LIN {X 0,Y 573.207,Z 132.087,A -85,B 0,C 180,E1 -2272.999,E2 -2272.999} C_VEL
LIN {X 0,Y 573.202,Z 132.089,A -85,B 0,C 180,E1 -2275.413,E2 -2275.413} C_VEL
LIN {X 0,Y 573.193,Z 132.083,A -85,B 0,C 180,E1 -2278.017,E2 -2278.017} C_VEL
LIN {X 0,Y 573.202,Z 132.084,A -85,B 0,C 180,E1 -2280.877,E2 -2280.877} C_VEL
LIN {X 0,Y 573.19,Z 132.087,A -85,B 0,C 180,E1 -2283.513,E2 -2283.513} C_VEL
LIN {X 0,Y 573.177,Z 132.082,A -85,B 0,C 180,E1 -2286.055,E2 -2286.055} C_VEL
LIN {X 0,Y 573.175,Z 132.086,A -85,B 0,C 180,E1 -2288.707,E2 -2288.707} C_VEL
LIN {X 0,Y 573.185,Z 132.084,A -85,B 0,C 180,E1 -2291.588,E2 -2291.588} C_VEL
LIN {X 0,Y 573.207,Z 132.08,A -85,B 0,C 180,E1 -2294.337,E2 -2294.337} C_VEL
LIN {X 0,Y 573.21,Z 132.082,A -85,B 0,C 180,E1 -2297.362,E2 -2297.362} C_VEL
LIN {X 0,Y 573.22,Z 132.081,A -85,B 0,C 180,E1 -2300.572,E2 -2300.572} C_VEL
LIN {X 0,Y 573.221,Z 132.083,A -85,B 0,C 180,E1 -2303.075,E2 -2303.075} C_VEL
LIN {X 0,Y 573.222,Z 132.077,A -85,B 0,C 180,E1 -2305.668,E2 -2305.668} C_VEL
LIN {X 0,Y 573.209,Z 132.079,A -85,B 0,C 180,E1 -2308.182,E2 -2308.182} C_VEL
LIN {X 0,Y 573.215,Z 132.086,A -85,B 0,C 180,E1 -2310.631,E2 -2310.631} C_VEL
LIN {X 0,Y 573.197,Z 132.08,A -85,B 0,C 180,E1 -2313.517,E2 -2313.517} C_VEL
LIN {X 0,Y 573.191,Z 132.082,A -85,B 0,C 180,E1 -2316.133,E2 -2316.133} C_VEL
LIN {X 0,Y 573.219,Z 132.077,A -85,B 0,C 180,E1 -2319.172,E2 -2319.172} C_VEL
LIN {X 0,Y 573.198,Z 132.084,A -85,B 0,C 180,E1 -2322.15,E2 -2322.15} C_VEL
LIN {X 0,Y 573.213,Z 132.078,A -85,B 0,C 180,E1 -2325.08,E2 -2325.08} C_VEL
LIN {X 0,Y 573.226,Z 132.079,A -85,B 0,C 180,E1 -2327.97,E2 -2327.97} C_VEL
LIN {X 0,Y 573.202,Z 132.084,A -85,B 0,C 180,E1 -2330.116,E2 -2330.116} C_VEL
LIN {X 0,Y 573.225,Z 132.076,A -85,B 0,C 180,E1 -2332.958,E2 -2332.958} C_VEL
LIN {X 0,Y 573.273,Z 132.07,A -85,B 0,C 180,E1 -2335.077,E2 -2335.077} C_VEL
LIN {X 0,Y 573.309,Z 132.07,A -85,B 0,C 180,E1 -2337.892,E2 -2337.892} C_VEL
LIN {X 0,Y 573.32,Z 132.071,A -85,B 0,C 180,E1 -2340,E2 -2340} C_VEL
LIN {X 0,Y 573.274,Z 132.071,A -85,B 0,C 180,E1 -2342.811,E2 -2342.811} C_VEL
LIN {X 0,Y 573.268,Z 132.074,A -85,B 0,C 180,E1 -2345.628,E2 -2345.628} C_VEL
LIN {X 0,Y 573.238,Z 132.077,A -85,B 0,C 180,E1 -2348.46,E2 -2348.46} C_VEL
LIN {X 0,Y 573.241,Z 132.076,A -85,B 0,C 180,E1 -2351.313,E2 -2351.313} C_VEL
LIN {X 0,Y 573.247,Z 132.076,A -85,B 0,C 180,E1 -2354.408,E2 -2354.408} C_VEL
LIN {X 0,Y 573.197,Z 132.081,A -85,B 0,C 180,E1 -2357.114,E2 -2357.114} C_VEL
LIN {X 0,Y 573.205,Z 132.083,A -85,B 0,C 180,E1 -2360.078,E2 -2360.078} C_VEL
LIN {X 0,Y 573.2,Z 132.081,A -85,B 0,C 180,E1 -2362.339,E2 -2362.339} C_VEL
LIN {X 0,Y 573.199,Z 132.081,A -85,B 0,C 180,E1 -2364.344,E2 -2364.344} C_VEL
LIN {X 0,Y 572.561,Z 132.161,A -85,B 0,C 180,E1 -2364.93,E2 -2364.93} C_VEL
LIN {X 0,Y 569.729,Z 132.519,A -85,B 0,C 180,E1 -2365.882,E2 -2365.882} C_VEL
LIN {X 0,Y 567.308,Z 132.823,A -85,B 0,C 180,E1 -2366.648,E2 -2366.648} C_VEL
LIN {X 0,Y 566.25,Z 132.952,A -85,B 0,C 180,E1 -2367.239,E2 -2367.239} C_VEL
LIN {X 0,Y 566.155,Z 132.962,A -85,B 0,C 180,E1 -2367.439,E2 -2367.439} C_VEL
LIN {X 0,Y 566.153,Z 132.964,A -85,B 0,C 180,E1 -2369.772,E2 -2369.772} C_VEL
LIN {X 0,Y 566.195,Z 132.953,A -85,B 0,C 180,E1 -2372.428,E2 -2372.428} C_VEL
LIN {X 0,Y 566.168,Z 132.959,A -85,B 0,C 180,E1 -2374.987,E2 -2374.987} C_VEL
LIN {X 0,Y 566.213,Z 132.958,A -85,B 0,C 180,E1 -2377.909,E2 -2377.909} C_VEL
LIN {X 0,Y 566.226,Z 133.057,A -85,B 0,C 180,E1 -2378.247,E2 -2378.247} C_VEL
LIN {X 0,Y 566.536,Z 138.801,A -85,B 0,C 180,E1 -2379.247,E2 -2379.247} C_VEL
LIN {X 0,Y 566.37,Z 154.943,A -85,B 0,C 180,E1 -2382.073,E2 -2382.073} C_VEL
LIN {X 0,Y 566.258,Z 166.155,A -85,B 0,C 180,E1 -2384.046,E2 -2384.046} C_VEL
LIN {X 0,Y 567.19,Z 172.386,A -85,B 0,C 180,E1 -2384.155,E2 -2384.155} C_VEL
LIN {X 0,Y 566.959,Z 273.025,A -85,B 0,C 180,E1 -2385.45,E2 -2385.45} C_VEL
LIN {X 0,Y 566.865,Z 286.291,A -85,B 0,C 180,E1 -2385.767,E2 -2385.767} C_VEL
LIN {X 0,Y 566.74,Z 298.58,A -85,B 0,C 180,E1 -2386.202,E2 -2386.202} C_VEL
LIN {X 0,Y 566.586,Z 310.977,A -85,B 0,C 180,E1 -2386.799,E2 -2386.799} C_VEL
LIN {X 0,Y 566.444,Z 321.518,A -85,B 0,C 180,E1 -2387.453,E2 -2387.453} C_VEL
LIN {X 0,Y 566.316,Z 331.988,A -85,B 0,C 180,E1 -2388.258,E2 -2388.258} C_VEL
LIN {X 0,Y 566.172,Z 340.62,A -85,B 0,C 180,E1 -2389.069,E2 -2389.069} C_VEL
LIN {X 0,Y 566.099,Z 349.526,A -85,B 0,C 180,E1 -2390.089,E2 -2390.089} C_VEL
LIN {X 0,Y 565.996,Z 356.78,A -85,B 0,C 180,E1 -2391.117,E2 -2391.117} C_VEL
LIN {X 0,Y 565.951,Z 363.434,A -85,B 0,C 180,E1 -2392.295,E2 -2392.295} C_VEL
LIN {X 0,Y 565.918,Z 368.346,A -85,B 0,C 180,E1 -2393.409,E2 -2393.409} C_VEL
LIN {X 0,Y 565.882,Z 372.568,A -85,B 0,C 180,E1 -2394.698,E2 -2394.698} C_VEL
LIN {X 0,Y 565.858,Z 375.371,A -85,B 0,C 180,E1 -2396.02,E2 -2396.02} C_VEL
LIN {X 0,Y 565.827,Z 376.461,A -85,B 0,C 180,E1 -2396.872,E2 -2396.872} C_VEL
LIN {X 0,Y 565.854,Z 376.934,A -85,B 0,C 180,E1 -2397.719,E2 -2397.719} C_VEL
LIN {X 0,Y 565.863,Z 376.636,A -85,B 0,C 180,E1 -2398.979,E2 -2398.979} C_VEL
LIN {X 0,Y 565.878,Z 374.842,A -85,B 0,C 180,E1 -2400.387,E2 -2400.387} C_VEL
LIN {X 0,Y 565.895,Z 372.452,A -85,B 0,C 180,E1 -2401.436,E2 -2401.436} C_VEL
LIN {X 0,Y 565.938,Z 368.487,A -85,B 0,C 180,E1 -2402.646,E2 -2402.646} C_VEL
LIN {X 0,Y 565.983,Z 363.185,A -85,B 0,C 180,E1 -2403.844,E2 -2403.844} C_VEL
LIN {X 0,Y 566,Z 356.44,A -85,B 0,C 180,E1 -2405.028,E2 -2405.028} C_VEL
LIN {X 0,Y 566.102,Z 349.461,A -85,B 0,C 180,E1 -2406.009,E2 -2406.009} C_VEL
LIN {X 0,Y 566.195,Z 340.847,A -85,B 0,C 180,E1 -2406.998,E2 -2406.998} C_VEL
LIN {X 0,Y 566.33,Z 330.572,A -85,B 0,C 180,E1 -2407.951,E2 -2407.951} C_VEL
LIN {X 0,Y 566.436,Z 320.727,A -85,B 0,C 180,E1 -2408.693,E2 -2408.693} C_VEL
LIN {X 0,Y 566.613,Z 309.091,A -85,B 0,C 180,E1 -2409.393,E2 -2409.393} C_VEL
LIN {X 0,Y 566.722,Z 296.67,A -85,B 0,C 180,E1 -2409.966,E2 -2409.966} C_VEL
LIN {X 0,Y 566.872,Z 283.539,A -85,B 0,C 180,E1 -2410.405,E2 -2410.405} C_VEL
LIN {X 0,Y 566.964,Z 270.481,A -85,B 0,C 180,E1 -2410.682,E2 -2410.682} C_VEL
LIN {X 0,Y 567.076,Z 171.372,A -85,B 0,C 180,E1 -2411.951,E2 -2411.951} C_VEL
LIN {X 0,Y 566.25,Z 166.047,A -85,B 0,C 180,E1 -2412.064,E2 -2412.064} C_VEL
LIN {X 0,Y 566.44,Z 149.983,A -85,B 0,C 180,E1 -2414.897,E2 -2414.897} C_VEL
LIN {X 0,Y 566.531,Z 135.544,A -85,B 0,C 180,E1 -2417.462,E2 -2417.462} C_VEL
LIN {X 0,Y 566.251,Z 132.952,A -85,B 0,C 180,E1 -2417.956,E2 -2417.956} C_VEL
LIN {X 0,Y 566.198,Z 132.961,A -85,B 0,C 180,E1 -2420.714,E2 -2420.714} C_VEL
LIN {X 0,Y 566.225,Z 132.95,A -85,B 0,C 180,E1 -2423.201,E2 -2423.201} C_VEL
LIN {X 0,Y 566.174,Z 132.955,A -85,B 0,C 180,E1 -2425.729,E2 -2425.729} C_VEL
LIN {X 0,Y 566.282,Z 132.943,A -85,B 0,C 180,E1 -2427.866,E2 -2427.866} C_VEL
LIN {X 0,Y 566.294,Z 132.944,A -85,B 0,C 180,E1 -2430.711,E2 -2430.711} C_VEL
LIN {X 0,Y 566.253,Z 132.947,A -85,B 0,C 180,E1 -2432.846,E2 -2432.846} C_VEL
LIN {X 0,Y 566.25,Z 132.947,A -85,B 0,C 180,E1 -2435.698,E2 -2435.698} C_VEL
LIN {X 0,Y 566.201,Z 132.955,A -85,B 0,C 180,E1 -2438.566,E2 -2438.566} C_VEL
LIN {X 0,Y 566.243,Z 132.947,A -85,B 0,C 180,E1 -2441.454,E2 -2441.454} C_VEL
LIN {X 0,Y 566.228,Z 132.95,A -85,B 0,C 180,E1 -2444.502,E2 -2444.502} C_VEL
LIN {X 0,Y 566.163,Z 132.957,A -85,B 0,C 180,E1 -2447.333,E2 -2447.333} C_VEL
LIN {X 0,Y 566.201,Z 132.956,A -85,B 0,C 180,E1 -2449.581,E2 -2449.581} C_VEL
LIN {X 0,Y 566.187,Z 132.963,A -85,B 0,C 180,E1 -2451.863,E2 -2451.863} C_VEL
LIN {X 0,Y 566.181,Z 132.954,A -85,B 0,C 180,E1 -2455.021,E2 -2455.021} C_VEL
LIN {X 0,Y 566.169,Z 132.959,A -85,B 0,C 180,E1 -2457.342,E2 -2457.342} C_VEL
LIN {X 0,Y 566.172,Z 132.963,A -85,B 0,C 180,E1 -2459.771,E2 -2459.771} C_VEL
LIN {X 0,Y 566.195,Z 132.952,A -85,B 0,C 180,E1 -2462.428,E2 -2462.428} C_VEL
LIN {X 0,Y 566.169,Z 132.957,A -85,B 0,C 180,E1 -2464.987,E2 -2464.987} C_VEL
LIN {X 0,Y 566.193,Z 132.962,A -85,B 0,C 180,E1 -2467.462,E2 -2467.462} C_VEL
LIN {X 0,Y 566.208,Z 132.95,A -85,B 0,C 180,E1 -2470.199,E2 -2470.199} C_VEL
LIN {X 0,Y 566.181,Z 132.959,A -85,B 0,C 180,E1 -2473.057,E2 -2473.057} C_VEL
LIN {X 0,Y 566.159,Z 132.957,A -85,B 0,C 180,E1 -2476.053,E2 -2476.053} C_VEL
LIN {X 0,Y 566.166,Z 132.96,A -85,B 0,C 180,E1 -2478.859,E2 -2478.859} C_VEL
LIN {X 0,Y 566.206,Z 132.955,A -85,B 0,C 180,E1 -2481.443,E2 -2481.443} C_VEL
LIN {X 0,Y 566.144,Z 132.959,A -85,B 0,C 180,E1 -2484.306,E2 -2484.306} C_VEL
LIN {X 0,Y 566.197,Z 132.96,A -85,B 0,C 180,E1 -2486.896,E2 -2486.896} C_VEL
LIN {X 0,Y 566.162,Z 132.959,A -85,B 0,C 180,E1 -2489.406,E2 -2489.406} C_VEL
LIN {X 0,Y 566.152,Z 132.957,A -85,B 0,C 180,E1 -2491.854,E2 -2491.854} C_VEL
LIN {X 0,Y 566.19,Z 132.954,A -85,B 0,C 180,E1 -2494.25,E2 -2494.25} C_VEL
LIN {X 0,Y 566.16,Z 132.966,A -85,B 0,C 180,E1 -2496.723,E2 -2496.723} C_VEL
LIN {X 0,Y 566.194,Z 132.958,A -85,B 0,C 180,E1 -2498.902,E2 -2498.902} C_VEL
LIN {X 0,Y 566.187,Z 132.955,A -85,B 0,C 180,E1 -2501.172,E2 -2501.172} C_VEL
LIN {X 0,Y 566.171,Z 132.958,A -85,B 0,C 180,E1 -2504.152,E2 -2504.152} C_VEL
LIN {X 0,Y 566.16,Z 132.963,A -85,B 0,C 180,E1 -2506.358,E2 -2506.358} C_VEL
LIN {X 0,Y 566.235,Z 132.947,A -85,B 0,C 180,E1 -2509.27,E2 -2509.27} C_VEL
LIN {X 0,Y 566.192,Z 132.958,A -85,B 0,C 180,E1 -2512.152,E2 -2512.152} C_VEL
LIN {X 0,Y 566.253,Z 132.945,A -85,B 0,C 180,E1 -2515.016,E2 -2515.016} C_VEL
LIN {X 0,Y 566.28,Z 132.945,A -85,B 0,C 180,E1 -2517.866,E2 -2517.866} C_VEL
LIN {X 0,Y 566.289,Z 132.947,A -85,B 0,C 180,E1 -2520,E2 -2520} C_VEL
LIN {X 0,Y 566.243,Z 132.946,A -85,B 0,C 180,E1 -2522.846,E2 -2522.846} C_VEL
LIN {X 0,Y 566.237,Z 132.951,A -85,B 0,C 180,E1 -2525.699,E2 -2525.699} C_VEL
LIN {X 0,Y 566.19,Z 132.954,A -85,B 0,C 180,E1 -2528.566,E2 -2528.566} C_VEL
LIN {X 0,Y 566.197,Z 132.954,A -85,B 0,C 180,E1 -2531.455,E2 -2531.455} C_VEL
LIN {X 0,Y 566.208,Z 132.951,A -85,B 0,C 180,E1 -2534.493,E2 -2534.493} C_VEL
LIN {X 0,Y 566.161,Z 132.959,A -85,B 0,C 180,E1 -2537.333,E2 -2537.333} C_VEL
LIN {X 0,Y 566.147,Z 132.959,A -85,B 0,C 180,E1 -2540.34,E2 -2540.34} C_VEL
LIN {X 0,Y 566.139,Z 132.959,A -85,B 0,C 180,E1 -2542.633,E2 -2542.633} C_VEL
LIN {X 0,Y 566.166,Z 132.957,A -85,B 0,C 180,E1 -2545.017,E2 -2545.017} C_VEL
LIN {X 0,Y 566.161,Z 132.963,A -85,B 0,C 180,E1 -2547.342,E2 -2547.342} C_VEL
LIN {X 0,Y 566.15,Z 132.962,A -85,B 0,C 180,E1 -2549.772,E2 -2549.772} C_VEL
LIN {X 0,Y 566.18,Z 132.954,A -85,B 0,C 180,E1 -2552.425,E2 -2552.425} C_VEL
LIN {X 0,Y 566.156,Z 132.961,A -85,B 0,C 180,E1 -2554.985,E2 -2554.985} C_VEL
LIN {X 0,Y 566.181,Z 132.96,A -85,B 0,C 180,E1 -2557.462,E2 -2557.462} C_VEL
LIN {X 0,Y 566.168,Z 132.955,A -85,B 0,C 180,E1 -2560.203,E2 -2560.203} C_VEL
LIN {X 0,Y 566.147,Z 132.966,A -85,B 0,C 180,E1 -2563.06,E2 -2563.06} C_VEL
LIN {X 0,Y 566.156,Z 132.956,A -85,B 0,C 180,E1 -2566.053,E2 -2566.053} C_VEL
LIN {X 0,Y 566.143,Z 132.966,A -85,B 0,C 180,E1 -2568.857,E2 -2568.857} C_VEL
LIN {X 0,Y 566.182,Z 132.956,A -85,B 0,C 180,E1 -2571.446,E2 -2571.446} C_VEL
LIN {X 0,Y 566.13,Z 132.962,A -85,B 0,C 180,E1 -2574.305,E2 -2574.305} C_VEL
LIN {X 0,Y 566.162,Z 132.964,A -85,B 0,C 180,E1 -2576.894,E2 -2576.894} C_VEL
LIN {X 0,Y 566.149,Z 132.959,A -85,B 0,C 180,E1 -2579.405,E2 -2579.405} C_VEL
LIN {X 0,Y 566.141,Z 132.96,A -85,B 0,C 180,E1 -2581.853,E2 -2581.853} C_VEL
LIN {X 0,Y 566.172,Z 132.96,A -85,B 0,C 180,E1 -2584.249,E2 -2584.249} C_VEL
LIN {X 0,Y 566.177,Z 133.142,A -85,B 0,C 180,E1 -2586.858,E2 -2586.858} C_VEL
LIN {X 0,Y 566.935,Z 139.049,A -85,B 0,C 180,E1 -2587.784,E2 -2587.784} C_VEL
LIN {X 0,Y 566.764,Z 157.831,A -85,B 0,C 180,E1 -2590.578,E2 -2590.578} C_VEL
LIN {X 0,Y 566.539,Z 177.246,A -85,B 0,C 180,E1 -2593.422,E2 -2593.422} C_VEL
LIN {X 0,Y 566.404,Z 195.133,A -85,B 0,C 180,E1 -2595.998,E2 -2595.998} C_VEL
LIN {X 0,Y 567.154,Z 200.499,A -85,B 0,C 180,E1 -2596.085,E2 -2596.085} C_VEL
LIN {X 0,Y 566.98,Z 302.941,A -85,B 0,C 180,E1 -2597.403,E2 -2597.403} C_VEL
LIN {X 0,Y 566.841,Z 316.214,A -85,B 0,C 180,E1 -2597.719,E2 -2597.719} C_VEL
LIN {X 0,Y 566.743,Z 328.375,A -85,B 0,C 180,E1 -2598.148,E2 -2598.148} C_VEL
LIN {X 0,Y 566.603,Z 340.363,A -85,B 0,C 180,E1 -2598.719,E2 -2598.719} C_VEL
LIN {X 0,Y 566.439,Z 352.194,A -85,B 0,C 180,E1 -2599.455,E2 -2599.455} C_VEL
LIN {X 0,Y 566.325,Z 362.603,A -85,B 0,C 180,E1 -2600.265,E2 -2600.265} C_VEL
LIN {X 0,Y 566.207,Z 371.112,A -85,B 0,C 180,E1 -2601.074,E2 -2601.074} C_VEL
LIN {X 0,Y 566.112,Z 378.96,A -85,B 0,C 180,E1 -2601.972,E2 -2601.972} C_VEL
LIN {X 0,Y 566.003,Z 386.622,A -85,B 0,C 180,E1 -2603.047,E2 -2603.047} C_VEL
LIN {X 0,Y 566.004,Z 393.679,A -85,B 0,C 180,E1 -2604.299,E2 -2604.299} C_VEL
LIN {X 0,Y 565.933,Z 398.372,A -85,B 0,C 180,E1 -2605.37,E2 -2605.37} C_VEL
LIN {X 0,Y 565.927,Z 401.958,A -85,B 0,C 180,E1 -2606.44,E2 -2606.44} C_VEL
LIN {X 0,Y 565.878,Z 403.807,A -85,B 0,C 180,E1 -2607.152,E2 -2607.152} C_VEL
LIN {X 0,Y 565.846,Z 406.184,A -85,B 0,C 180,E1 -2608.577,E2 -2608.577} C_VEL
LIN {X 0,Y 565.839,Z 407,A -85,B 0,C 180,E1 -2610,E2 -2610} C_VEL
LIN {X 0,Y 565.846,Z 406.185,A -85,B 0,C 180,E1 -2611.423,E2 -2611.423} C_VEL
LIN {X 0,Y 565.878,Z 403.81,A -85,B 0,C 180,E1 -2612.848,E2 -2612.848} C_VEL
LIN {X 0,Y 565.926,Z 400.895,A -85,B 0,C 180,E1 -2613.917,E2 -2613.917} C_VEL
LIN {X 0,Y 565.878,Z 396.948,A -85,B 0,C 180,E1 -2614.988,E2 -2614.988} C_VEL
LIN {X 0,Y 566.002,Z 391.867,A -85,B 0,C 180,E1 -2616.059,E2 -2616.059} C_VEL
LIN {X 0,Y 566.04,Z 385.467,A -85,B 0,C 180,E1 -2617.132,E2 -2617.132} C_VEL
LIN {X 0,Y 566.134,Z 377.477,A -85,B 0,C 180,E1 -2618.208,E2 -2618.208} C_VEL
LIN {X 0,Y 566.229,Z 369.333,A -85,B 0,C 180,E1 -2619.106,E2 -2619.106} C_VEL
LIN {X 0,Y 566.347,Z 359.397,A -85,B 0,C 180,E1 -2620.005,E2 -2620.005} C_VEL
LIN {X 0,Y 566.536,Z 348.289,A -85,B 0,C 180,E1 -2620.807,E2 -2620.807} C_VEL
LIN {X 0,Y 566.613,Z 337.17,A -85,B 0,C 180,E1 -2621.447,E2 -2621.447} C_VEL
LIN {X 0,Y 566.745,Z 324.975,A -85,B 0,C 180,E1 -2621.988,E2 -2621.988} C_VEL
LIN {X 0,Y 566.917,Z 312.168,A -85,B 0,C 180,E1 -2622.393,E2 -2622.393} C_VEL
LIN {X 0,Y 566.994,Z 300.095,A -85,B 0,C 180,E1 -2622.642,E2 -2622.642} C_VEL
LIN {X 0,Y 567.043,Z 199.378,A -85,B 0,C 180,E1 -2623.932,E2 -2623.932} C_VEL
LIN {X 0,Y 566.384,Z 194.791,A -85,B 0,C 180,E1 -2624.026,E2 -2624.026} C_VEL
LIN {X 0,Y 566.551,Z 175.036,A -85,B 0,C 180,E1 -2626.896,E2 -2626.896} C_VEL
LIN {X 0,Y 566.754,Z 156.798,A -85,B 0,C 180,E1 -2629.561,E2 -2629.561} C_VEL
LIN {X 0,Y 566.92,Z 138.88,A -85,B 0,C 180,E1 -2632.216,E2 -2632.216} C_VEL
LIN {X 0,Y 566.173,Z 133.051,A -85,B 0,C 180,E1 -2633.117,E2 -2633.117} C_VEL
LIN {X 0,Y 566.172,Z 132.96,A -85,B 0,C 180,E1 -2635.751,E2 -2635.751} C_VEL
LIN {X 0,Y 566.138,Z 132.961,A -85,B 0,C 180,E1 -2638.189,E2 -2638.189} C_VEL
LIN {X 0,Y 566.17,Z 132.963,A -85,B 0,C 180,E1 -2641.072,E2 -2641.072} C_VEL
LIN {X 0,Y 566.16,Z 132.96,A -85,B 0,C 180,E1 -2643.726,E2 -2643.726} C_VEL
LIN {X 0,Y 566.14,Z 132.961,A -85,B 0,C 180,E1 -2646.575,E2 -2646.575} C_VEL
LIN {X 0,Y 566.177,Z 132.957,A -85,B 0,C 180,E1 -2649.681,E2 -2649.681} C_VEL
LIN {X 0,Y 566.148,Z 132.965,A -85,B 0,C 180,E1 -2652.911,E2 -2652.911} C_VEL
LIN {X 0,Y 566.149,Z 132.958,A -85,B 0,C 180,E1 -2655.959,E2 -2655.959} C_VEL
LIN {X 0,Y 566.139,Z 132.968,A -85,B 0,C 180,E1 -2658.857,E2 -2658.857} C_VEL
LIN {X 0,Y 566.158,Z 132.959,A -85,B 0,C 180,E1 -2661.449,E2 -2661.449} C_VEL
LIN {X 0,Y 566.155,Z 132.956,A -85,B 0,C 180,E1 -2663.793,E2 -2663.793} C_VEL
LIN {X 0,Y 566.162,Z 132.958,A -85,B 0,C 180,E1 -2666.274,E2 -2666.274} C_VEL
LIN {X 0,Y 566.171,Z 132.962,A -85,B 0,C 180,E1 -2668.928,E2 -2668.928} C_VEL
LIN {X 0,Y 566.142,Z 132.958,A -85,B 0,C 180,E1 -2671.854,E2 -2671.854} C_VEL
LIN {X 0,Y 566.174,Z 132.958,A -85,B 0,C 180,E1 -2674.249,E2 -2674.249} C_VEL
LIN {X 0,Y 566.15,Z 132.965,A -85,B 0,C 180,E1 -2676.725,E2 -2676.725} C_VEL
LIN {X 0,Y 566.185,Z 132.956,A -85,B 0,C 180,E1 -2678.901,E2 -2678.901} C_VEL
LIN {X 0,Y 566.153,Z 132.959,A -85,B 0,C 180,E1 -2681.92,E2 -2681.92} C_VEL
LIN {X 0,Y 566.156,Z 132.959,A -85,B 0,C 180,E1 -2684.889,E2 -2684.889} C_VEL
LIN {X 0,Y 566.165,Z 132.957,A -85,B 0,C 180,E1 -2687.817,E2 -2687.817} C_VEL
LIN {X 0,Y 566.157,Z 132.959,A -85,B 0,C 180,E1 -2689.992,E2 -2689.992} C_VEL
LIN {X 0,Y 566.187,Z 132.953,A -85,B 0,C 180,E1 -2692.87,E2 -2692.87} C_VEL
LIN {X 0,Y 566.25,Z 132.945,A -85,B 0,C 180,E1 -2695.016,E2 -2695.016} C_VEL
LIN {X 0,Y 566.279,Z 132.945,A -85,B 0,C 180,E1 -2697.866,E2 -2697.866} C_VEL
LIN {X 0,Y 566.289,Z 132.947,A -85,B 0,C 180,E1 -2700,E2 -2700} C_VEL
LIN {X 0,Y 566.241,Z 132.946,A -85,B 0,C 180,E1 -2702.846,E2 -2702.846} C_VEL
LIN {X 0,Y 566.237,Z 132.951,A -85,B 0,C 180,E1 -2705.699,E2 -2705.699} C_VEL
LIN {X 0,Y 566.19,Z 132.954,A -85,B 0,C 180,E1 -2708.566,E2 -2708.566} C_VEL
LIN {X 0,Y 566.198,Z 132.955,A -85,B 0,C 180,E1 -2711.455,E2 -2711.455} C_VEL
LIN {X 0,Y 566.208,Z 132.952,A -85,B 0,C 180,E1 -2714.493,E2 -2714.493} C_VEL
LIN {X 0,Y 566.162,Z 132.959,A -85,B 0,C 180,E1 -2717.333,E2 -2717.333} C_VEL
LIN {X 0,Y 566.177,Z 132.961,A -85,B 0,C 180,E1 -2719.582,E2 -2719.582} C_VEL
LIN {X 0,Y 566.151,Z 132.965,A -85,B 0,C 180,E1 -2721.864,E2 -2721.864} C_VEL
LIN {X 0,Y 566.199,Z 132.953,A -85,B 0,C 180,E1 -2724.963,E2 -2724.963} C_VEL
LIN {X 0,Y 566.155,Z 132.962,A -85,B 0,C 180,E1 -2727.439,E2 -2727.439} C_VEL
LIN {X 0,Y 565.46,Z 133.048,A -85,B 0,C 180,E1 -2728.033,E2 -2728.033} C_VEL
LIN {X 0,Y 562.586,Z 133.404,A -85,B 0,C 180,E1 -2728.997,E2 -2728.997} C_VEL
LIN {X 0,Y 560.186,Z 133.708,A -85,B 0,C 180,E1 -2729.772,E2 -2729.772} C_VEL
LIN {X 0,Y 559.177,Z 133.828,A -85,B 0,C 180,E1 -2730.371,E2 -2730.371} C_VEL
LIN {X 0,Y 559.105,Z 133.836,A -85,B 0,C 180,E1 -2730.574,E2 -2730.574} C_VEL
LIN {X 0,Y 559.151,Z 133.831,A -85,B 0,C 180,E1 -2732.716,E2 -2732.716} C_VEL
LIN {X 0,Y 559.119,Z 133.842,A -85,B 0,C 180,E1 -2735.325,E2 -2735.325} C_VEL
LIN {X 0,Y 559.18,Z 133.921,A -85,B 0,C 180,E1 -2738.157,E2 -2738.157} C_VEL
LIN {X 0,Y 559.541,Z 139.473,A -85,B 0,C 180,E1 -2739.136,E2 -2739.136} C_VEL
LIN {X 0,Y 559.371,Z 155.496,A -85,B 0,C 180,E1 -2741.954,E2 -2741.954} C_VEL
LIN {X 0,Y 559.222,Z 166.248,A -85,B 0,C 180,E1 -2743.87,E2 -2743.87} C_VEL
LIN {X 0,Y 560.305,Z 173.003,A -85,B 0,C 180,E1 -2743.988,E2 -2743.988} C_VEL
LIN {X 0,Y 560.036,Z 273.461,A -85,B 0,C 180,E1 -2745.3,E2 -2745.3} C_VEL
LIN {X 0,Y 559.929,Z 287.105,A -85,B 0,C 180,E1 -2745.636,E2 -2745.636} C_VEL
LIN {X 0,Y 559.77,Z 299.441,A -85,B 0,C 180,E1 -2746.087,E2 -2746.087} C_VEL
LIN {X 0,Y 559.598,Z 311.663,A -85,B 0,C 180,E1 -2746.697,E2 -2746.697} C_VEL
LIN {X 0,Y 559.429,Z 323.258,A -85,B 0,C 180,E1 -2747.442,E2 -2747.442} C_VEL
LIN {X 0,Y 559.294,Z 333.235,A -85,B 0,C 180,E1 -2748.241,E2 -2748.241} C_VEL
LIN {X 0,Y 559.093,Z 342.738,A -85,B 0,C 180,E1 -2749.182,E2 -2749.182} C_VEL
LIN {X 0,Y 559.041,Z 350.526,A -85,B 0,C 180,E1 -2750.122,E2 -2750.122} C_VEL
LIN {X 0,Y 558.911,Z 357.993,A -85,B 0,C 180,E1 -2751.226,E2 -2751.226} C_VEL
LIN {X 0,Y 558.879,Z 364.294,A -85,B 0,C 180,E1 -2752.395,E2 -2752.395} C_VEL
LIN {X 0,Y 558.849,Z 369.846,A -85,B 0,C 180,E1 -2753.767,E2 -2753.767} C_VEL
LIN {X 0,Y 558.786,Z 373.018,A -85,B 0,C 180,E1 -2754.838,E2 -2754.838} C_VEL
LIN {X 0,Y 558.762,Z 375.555,A -85,B 0,C 180,E1 -2756.113,E2 -2756.113} C_VEL
LIN {X 0,Y 558.756,Z 376.853,A -85,B 0,C 180,E1 -2757.429,E2 -2757.429} C_VEL
LIN {X 0,Y 558.761,Z 376.768,A -85,B 0,C 180,E1 -2758.792,E2 -2758.792} C_VEL
LIN {X 0,Y 558.767,Z 375.188,A -85,B 0,C 180,E1 -2760.211,E2 -2760.211} C_VEL
LIN {X 0,Y 558.793,Z 371.839,A -85,B 0,C 180,E1 -2761.691,E2 -2761.691} C_VEL
LIN {X 0,Y 558.848,Z 367.007,A -85,B 0,C 180,E1 -2763.081,E2 -2763.081} C_VEL
LIN {X 0,Y 558.92,Z 361.274,A -85,B 0,C 180,E1 -2764.29,E2 -2764.29} C_VEL
LIN {X 0,Y 558.969,Z 353.989,A -85,B 0,C 180,E1 -2765.486,E2 -2765.486} C_VEL
LIN {X 0,Y 559.107,Z 345.65,A -85,B 0,C 180,E1 -2766.58,E2 -2766.58} C_VEL
LIN {X 0,Y 559.252,Z 336.347,A -85,B 0,C 180,E1 -2767.56,E2 -2767.56} C_VEL
LIN {X 0,Y 559.401,Z 325.498,A -85,B 0,C 180,E1 -2768.482,E2 -2768.482} C_VEL
LIN {X 0,Y 559.591,Z 314.667,A -85,B 0,C 180,E1 -2769.219,E2 -2769.219} C_VEL
LIN {X 0,Y 559.759,Z 302.814,A -85,B 0,C 180,E1 -2769.849,E2 -2769.849} C_VEL
LIN {X 0,Y 559.855,Z 291.656,A -85,B 0,C 180,E1 -2770.305,E2 -2770.305} C_VEL
LIN {X 0,Y 560.002,Z 278.619,A -85,B 0,C 180,E1 -2770.684,E2 -2770.684} C_VEL
LIN {X 0,Y 560.063,Z 265.242,A -85,B 0,C 180,E1 -2770.916,E2 -2770.916} C_VEL
LIN {X 0,Y 560.257,Z 172.606,A -85,B 0,C 180,E1 -2772.108,E2 -2772.108} C_VEL
LIN {X 0,Y 559.256,Z 166.202,A -85,B 0,C 180,E1 -2772.228,E2 -2772.228} C_VEL
LIN {X 0,Y 559.465,Z 149.022,A -85,B 0,C 180,E1 -2775.302,E2 -2775.302} C_VEL
LIN {X 0,Y 559.547,Z 136.837,A -85,B 0,C 180,E1 -2777.487,E2 -2777.487} C_VEL
LIN {X 0,Y 559.204,Z 133.831,A -85,B 0,C 180,E1 -2778.078,E2 -2778.078} C_VEL
LIN {X 0,Y 559.166,Z 133.83,A -85,B 0,C 180,E1 -2781.325,E2 -2781.325} C_VEL
LIN {X 0,Y 559.22,Z 133.827,A -85,B 0,C 180,E1 -2784.23,E2 -2784.23} C_VEL
LIN {X 0,Y 559.253,Z 133.818,A -85,B 0,C 180,E1 -2787.839,E2 -2787.839} C_VEL
LIN {X 0,Y 559.266,Z 133.819,A -85,B 0,C 180,E1 -2790.72,E2 -2790.72} C_VEL
LIN {X 0,Y 559.22,Z 133.822,A -85,B 0,C 180,E1 -2792.881,E2 -2792.881} C_VEL
LIN {X 0,Y 559.219,Z 133.824,A -85,B 0,C 180,E1 -2795.77,E2 -2795.77} C_VEL
LIN {X 0,Y 559.165,Z 133.83,A -85,B 0,C 180,E1 -2798.675,E2 -2798.675} C_VEL
LIN {X 0,Y 559.204,Z 133.825,A -85,B 0,C 180,E1 -2801.601,E2 -2801.601} C_VEL
LIN {X 0,Y 559.184,Z 133.827,A -85,B 0,C 180,E1 -2804.588,E2 -2804.588} C_VEL
LIN {X 0,Y 559.118,Z 133.837,A -85,B 0,C 180,E1 -2807.558,E2 -2807.558} C_VEL
LIN {X 0,Y 559.163,Z 133.837,A -85,B 0,C 180,E1 -2809.838,E2 -2809.838} C_VEL
LIN {X 0,Y 559.133,Z 133.836,A -85,B 0,C 180,E1 -2812.153,E2 -2812.153} C_VEL
LIN {X 0,Y 559.142,Z 133.832,A -85,B 0,C 180,E1 -2815.178,E2 -2815.178} C_VEL
LIN {X 0,Y 559.111,Z 133.844,A -85,B 0,C 180,E1 -2817.716,E2 -2817.716} C_VEL
LIN {X 0,Y 559.138,Z 133.833,A -85,B 0,C 180,E1 -2820.184,E2 -2820.184} C_VEL
LIN {X 0,Y 559.15,Z 133.829,A -85,B 0,C 180,E1 -2822.716,E2 -2822.716} C_VEL
LIN {X 0,Y 559.119,Z 133.84,A -85,B 0,C 180,E1 -2825.325,E2 -2825.325} C_VEL
LIN {X 0,Y 559.129,Z 133.834,A -85,B 0,C 180,E1 -2828.018,E2 -2828.018} C_VEL
LIN {X 0,Y 559.156,Z 133.83,A -85,B 0,C 180,E1 -2830.813,E2 -2830.813} C_VEL
LIN {X 0,Y 559.11,Z 133.838,A -85,B 0,C 180,E1 -2833.737,E2 -2833.737} C_VEL
LIN {X 0,Y 559.11,Z 133.834,A -85,B 0,C 180,E1 -2836.263,E2 -2836.263} C_VEL
LIN {X 0,Y 559.156,Z 133.839,A -85,B 0,C 180,E1 -2839.187,E2 -2839.187} C_VEL
LIN {X 0,Y 559.129,Z 133.832,A -85,B 0,C 180,E1 -2841.982,E2 -2841.982} C_VEL
LIN {X 0,Y 559.125,Z 133.838,A -85,B 0,C 180,E1 -2844.789,E2 -2844.789} C_VEL
LIN {X 0,Y 559.152,Z 133.833,A -85,B 0,C 180,E1 -2847.366,E2 -2847.366} C_VEL
LIN {X 0,Y 559.113,Z 133.835,A -85,B 0,C 180,E1 -2850.15,E2 -2850.15} C_VEL
LIN {X 0,Y 559.126,Z 133.837,A -85,B 0,C 180,E1 -2853.183,E2 -2853.183} C_VEL
LIN {X 0,Y 559.109,Z 133.835,A -85,B 0,C 180,E1 -2855.493,E2 -2855.493} C_VEL
LIN {X 0,Y 559.163,Z 133.836,A -85,B 0,C 180,E1 -2858.623,E2 -2858.623} C_VEL
LIN {X 0,Y 559.158,Z 133.834,A -85,B 0,C 180,E1 -2860.926,E2 -2860.926} C_VEL
LIN {X 0,Y 559.128,Z 133.833,A -85,B 0,C 180,E1 -2863.947,E2 -2863.947} C_VEL
LIN {X 0,Y 559.138,Z 133.835,A -85,B 0,C 180,E1 -2866.183,E2 -2866.183} C_VEL
LIN {X 0,Y 559.194,Z 133.825,A -85,B 0,C 180,E1 -2869.133,E2 -2869.133} C_VEL
LIN {X 0,Y 559.144,Z 133.835,A -85,B 0,C 180,E1 -2872.053,E2 -2872.053} C_VEL
LIN {X 0,Y 559.23,Z 133.821,A -85,B 0,C 180,E1 -2874.953,E2 -2874.953} C_VEL
LIN {X 0,Y 559.25,Z 133.82,A -85,B 0,C 180,E1 -2877.839,E2 -2877.839} C_VEL
LIN {X 0,Y 559.257,Z 133.823,A -85,B 0,C 180,E1 -2880,E2 -2880} C_VEL
LIN {X 0,Y 559.211,Z 133.822,A -85,B 0,C 180,E1 -2882.882,E2 -2882.882} C_VEL
LIN {X 0,Y 559.206,Z 133.828,A -85,B 0,C 180,E1 -2885.77,E2 -2885.77} C_VEL
LIN {X 0,Y 559.155,Z 133.83,A -85,B 0,C 180,E1 -2888.675,E2 -2888.675} C_VEL
LIN {X 0,Y 559.158,Z 133.833,A -85,B 0,C 180,E1 -2891.601,E2 -2891.601} C_VEL
LIN {X 0,Y 559.157,Z 133.829,A -85,B 0,C 180,E1 -2894.576,E2 -2894.576} C_VEL
LIN {X 0,Y 559.113,Z 133.84,A -85,B 0,C 180,E1 -2897.558,E2 -2897.558} C_VEL
LIN {X 0,Y 559.11,Z 133.834,A -85,B 0,C 180,E1 -2900.607,E2 -2900.607} C_VEL
LIN {X 0,Y 559.1,Z 133.842,A -85,B 0,C 180,E1 -2903.418,E2 -2903.418} C_VEL
LIN {X 0,Y 559.15,Z 133.831,A -85,B 0,C 180,E1 -2906.099,E2 -2906.099} C_VEL
LIN {X 0,Y 559.102,Z 133.835,A -85,B 0,C 180,E1 -2908.533,E2 -2908.533} C_VEL
LIN {X 0,Y 559.121,Z 133.84,A -85,B 0,C 180,E1 -2911.268,E2 -2911.268} C_VEL
LIN {X 0,Y 559.14,Z 133.832,A -85,B 0,C 180,E1 -2913.944,E2 -2913.944} C_VEL
LIN {X 0,Y 559.113,Z 133.841,A -85,B 0,C 180,E1 -2917.111,E2 -2917.111} C_VEL
LIN {X 0,Y 559.127,Z 133.833,A -85,B 0,C 180,E1 -2919.937,E2 -2919.937} C_VEL
LIN {X 0,Y 559.113,Z 133.838,A -85,B 0,C 180,E1 -2922.748,E2 -2922.748} C_VEL
LIN {X 0,Y 559.125,Z 133.833,A -85,B 0,C 180,E1 -2925.764,E2 -2925.764} C_VEL
LIN {X 0,Y 559.098,Z 133.836,A -85,B 0,C 180,E1 -2928.223,E2 -2928.223} C_VEL
LIN {X 0,Y 559.136,Z 133.837,A -85,B 0,C 180,E1 -2931.197,E2 -2931.197} C_VEL
LIN {X 0,Y 559.109,Z 133.834,A -85,B 0,C 180,E1 -2933.787,E2 -2933.787} C_VEL
LIN {X 0,Y 559.124,Z 133.836,A -85,B 0,C 180,E1 -2936.422,E2 -2936.422} C_VEL
LIN {X 0,Y 559.135,Z 133.838,A -85,B 0,C 180,E1 -2938.979,E2 -2938.979} C_VEL
LIN {X 0,Y 559.103,Z 133.836,A -85,B 0,C 180,E1 -2941.632,E2 -2941.632} C_VEL
LIN {X 0,Y 559.142,Z 133.833,A -85,B 0,C 180,E1 -2943.901,E2 -2943.901} C_VEL
LIN {X 0,Y 559.117,Z 133.925,A -85,B 0,C 180,E1 -2946.694,E2 -2946.694} C_VEL
LIN {X 0,Y 559.997,Z 140.166,A -85,B 0,C 180,E1 -2947.688,E2 -2947.688} C_VEL
LIN {X 0,Y 559.791,Z 158.413,A -85,B 0,C 180,E1 -2950.44,E2 -2950.44} C_VEL
LIN {X 0,Y 559.526,Z 177.076,A -85,B 0,C 180,E1 -2953.208,E2 -2953.208} C_VEL
LIN {X 0,Y 559.388,Z 194.976,A -85,B 0,C 180,E1 -2955.818,E2 -2955.818} C_VEL
LIN {X 0,Y 560.268,Z 202.176,A -85,B 0,C 180,E1 -2955.934,E2 -2955.934} C_VEL
LIN {X 0,Y 560.073,Z 302.94,A -85,B 0,C 180,E1 -2957.245,E2 -2957.245} C_VEL
LIN {X 0,Y 559.916,Z 316.213,A -85,B 0,C 180,E1 -2957.564,E2 -2957.564} C_VEL
LIN {X 0,Y 559.792,Z 328.374,A -85,B 0,C 180,E1 -2957.999,E2 -2957.999} C_VEL
LIN {X 0,Y 559.629,Z 340.191,A -85,B 0,C 180,E1 -2958.567,E2 -2958.567} C_VEL
LIN {X 0,Y 559.458,Z 352.192,A -85,B 0,C 180,E1 -2959.322,E2 -2959.322} C_VEL
LIN {X 0,Y 559.305,Z 362.604,A -85,B 0,C 180,E1 -2960.142,E2 -2960.142} C_VEL
LIN {X 0,Y 559.162,Z 371.113,A -85,B 0,C 180,E1 -2960.961,E2 -2960.961} C_VEL
LIN {X 0,Y 559.05,Z 378.96,A -85,B 0,C 180,E1 -2961.869,E2 -2961.869} C_VEL
LIN {X 0,Y 558.944,Z 386.622,A -85,B 0,C 180,E1 -2962.958,E2 -2962.958} C_VEL
LIN {X 0,Y 558.936,Z 393.679,A -85,B 0,C 180,E1 -2964.227,E2 -2964.227} C_VEL
LIN {X 0,Y 558.826,Z 398.373,A -85,B 0,C 180,E1 -2965.311,E2 -2965.311} C_VEL
LIN {X 0,Y 558.836,Z 401.958,A -85,B 0,C 180,E1 -2966.395,E2 -2966.395} C_VEL
LIN {X 0,Y 558.799,Z 403.807,A -85,B 0,C 180,E1 -2967.116,E2 -2967.116} C_VEL
LIN {X 0,Y 558.745,Z 406.183,A -85,B 0,C 180,E1 -2968.558,E2 -2968.558} C_VEL
LIN {X 0,Y 558.74,Z 407,A -85,B 0,C 180,E1 -2970,E2 -2970} C_VEL
LIN {X 0,Y 558.745,Z 406.184,A -85,B 0,C 180,E1 -2971.442,E2 -2971.442} C_VEL
LIN {X 0,Y 558.799,Z 403.81,A -85,B 0,C 180,E1 -2972.884,E2 -2972.884} C_VEL
LIN {X 0,Y 558.844,Z 400.895,A -85,B 0,C 180,E1 -2973.966,E2 -2973.966} C_VEL
LIN {X 0,Y 558.798,Z 396.948,A -85,B 0,C 180,E1 -2975.051,E2 -2975.051} C_VEL
LIN {X 0,Y 558.922,Z 391.867,A -85,B 0,C 180,E1 -2976.136,E2 -2976.136} C_VEL
LIN {X 0,Y 558.977,Z 385.466,A -85,B 0,C 180,E1 -2977.223,E2 -2977.223} C_VEL
LIN {X 0,Y 559.099,Z 377.476,A -85,B 0,C 180,E1 -2978.312,E2 -2978.312} C_VEL
LIN {X 0,Y 559.195,Z 369.332,A -85,B 0,C 180,E1 -2979.221,E2 -2979.221} C_VEL
LIN {X 0,Y 559.357,Z 359.396,A -85,B 0,C 180,E1 -2980.131,E2 -2980.131} C_VEL
LIN {X 0,Y 559.556,Z 348.395,A -85,B 0,C 180,E1 -2980.937,E2 -2980.937} C_VEL
LIN {X 0,Y 559.672,Z 336.454,A -85,B 0,C 180,E1 -2981.628,E2 -2981.628} C_VEL
LIN {X 0,Y 559.822,Z 324.972,A -85,B 0,C 180,E1 -2982.139,E2 -2982.139} C_VEL
LIN {X 0,Y 559.982,Z 312.167,A -85,B 0,C 180,E1 -2982.549,E2 -2982.549} C_VEL
LIN {X 0,Y 560.088,Z 298.584,A -85,B 0,C 180,E1 -2982.823,E2 -2982.823} C_VEL
LIN {X 0,Y 560.202,Z 200.359,A -85,B 0,C 180,E1 -2984.091,E2 -2984.091} C_VEL
LIN {X 0,Y 559.368,Z 194.675,A -85,B 0,C 180,E1 -2984.205,E2 -2984.205} C_VEL
LIN {X 0,Y 559.526,Z 175.156,A -85,B 0,C 180,E1 -2987.063,E2 -2987.063} C_VEL
LIN {X 0,Y 559.769,Z 157.537,A -85,B 0,C 180,E1 -2989.671,E2 -2989.671} C_VEL
LIN {X 0,Y 559.977,Z 139.922,A -85,B 0,C 180,E1 -2992.312,E2 -2992.312} C_VEL
LIN {X 0,Y 559.12,Z 133.843,A -85,B 0,C 180,E1 -2993.277,E2 -2993.277} C_VEL
LIN {X 0,Y 559.141,Z 133.833,A -85,B 0,C 180,E1 -2996.099,E2 -2996.099} C_VEL
LIN {X 0,Y 559.099,Z 133.838,A -85,B 0,C 180,E1 -2998.534,E2 -2998.534} C_VEL
LIN {X 0,Y 559.117,Z 133.844,A -85,B 0,C 180,E1 -3001.268,E2 -3001.268} C_VEL
LIN {X 0,Y 559.125,Z 133.835,A -85,B 0,C 180,E1 -3003.942,E2 -3003.942} C_VEL
LIN {X 0,Y 559.097,Z 133.837,A -85,B 0,C 180,E1 -3006.438,E2 -3006.438} C_VEL
LIN {X 0,Y 559.125,Z 133.84,A -85,B 0,C 180,E1 -3008.939,E2 -3008.939} C_VEL
LIN {X 0,Y 559.111,Z 133.835,A -85,B 0,C 180,E1 -3012.13,E2 -3012.13} C_VEL
LIN {X 0,Y 559.122,Z 133.84,A -85,B 0,C 180,E1 -3015.259,E2 -3015.259} C_VEL
LIN {X 0,Y 559.096,Z 133.837,A -85,B 0,C 180,E1 -3018.223,E2 -3018.223} C_VEL
LIN {X 0,Y 559.125,Z 133.84,A -85,B 0,C 180,E1 -3021.062,E2 -3021.062} C_VEL
LIN {X 0,Y 559.11,Z 133.834,A -85,B 0,C 180,E1 -3023.787,E2 -3023.787} C_VEL
LIN {X 0,Y 559.107,Z 133.839,A -85,B 0,C 180,E1 -3026.421,E2 -3026.421} C_VEL
LIN {X 0,Y 559.137,Z 133.837,A -85,B 0,C 180,E1 -3028.979,E2 -3028.979} C_VEL
LIN {X 0,Y 559.105,Z 133.834,A -85,B 0,C 180,E1 -3031.632,E2 -3031.632} C_VEL
LIN {X 0,Y 559.144,Z 133.831,A -85,B 0,C 180,E1 -3033.901,E2 -3033.901} C_VEL
LIN {X 0,Y 559.094,Z 133.839,A -85,B 0,C 180,E1 -3037.065,E2 -3037.065} C_VEL
LIN {X 0,Y 559.108,Z 133.833,A -85,B 0,C 180,E1 -3039.393,E2 -3039.393} C_VEL
LIN {X 0,Y 559.112,Z 133.843,A -85,B 0,C 180,E1 -3042.442,E2 -3042.442} C_VEL
LIN {X 0,Y 559.156,Z 133.828,A -85,B 0,C 180,E1 -3045.441,E2 -3045.441} C_VEL
LIN {X 0,Y 559.15,Z 133.833,A -85,B 0,C 180,E1 -3048.637,E2 -3048.637} C_VEL
LIN {X 0,Y 559.152,Z 133.829,A -85,B 0,C 180,E1 -3051.325,E2 -3051.325} C_VEL
LIN {X 0,Y 559.206,Z 133.83,A -85,B 0,C 180,E1 -3054.23,E2 -3054.23} C_VEL
LIN {X 0,Y 559.25,Z 133.82,A -85,B 0,C 180,E1 -3057.839,E2 -3057.839} C_VEL
LIN {X 0,Y 559.257,Z 133.823,A -85,B 0,C 180,E1 -3060,E2 -3060} C_VEL
LIN {X 0,Y 559.209,Z 133.822,A -85,B 0,C 180,E1 -3062.882,E2 -3062.882} C_VEL
LIN {X 0,Y 559.206,Z 133.828,A -85,B 0,C 180,E1 -3065.77,E2 -3065.77} C_VEL
LIN {X 0,Y 559.155,Z 133.829,A -85,B 0,C 180,E1 -3068.675,E2 -3068.675} C_VEL
LIN {X 0,Y 559.16,Z 133.833,A -85,B 0,C 180,E1 -3071.601,E2 -3071.601} C_VEL
LIN {X 0,Y 559.158,Z 133.83,A -85,B 0,C 180,E1 -3074.576,E2 -3074.576} C_VEL
LIN {X 0,Y 559.115,Z 133.84,A -85,B 0,C 180,E1 -3077.558,E2 -3077.558} C_VEL
LIN {X 0,Y 559.14,Z 133.839,A -85,B 0,C 180,E1 -3079.839,E2 -3079.839} C_VEL
LIN {X 0,Y 559.107,Z 133.839,A -85,B 0,C 180,E1 -3082.154,E2 -3082.154} C_VEL
LIN {X 0,Y 559.143,Z 133.834,A -85,B 0,C 180,E1 -3085.178,E2 -3085.178} C_VEL
LIN {X 0,Y 559.105,Z 133.844,A -85,B 0,C 180,E1 -3087.716,E2 -3087.716} C_VEL
LIN {X 0,Y 559.105,Z 133.836,A -85,B 0,C 180,E1 -3090.574,E2 -3090.574} C_VEL
LIN {X 0,Y 558.465,Z 133.921,A -85,B 0,C 180,E1 -3091.176,E2 -3091.176} C_VEL
LIN {X 0,Y 555.617,Z 134.272,A -85,B 0,C 180,E1 -3092.152,E2 -3092.152} C_VEL
LIN {X 0,Y 553.199,Z 134.574,A -85,B 0,C 180,E1 -3092.938,E2 -3092.938} C_VEL
LIN {X 0,Y 552.168,Z 134.709,A -85,B 0,C 180,E1 -3093.545,E2 -3093.545} C_VEL
LIN {X 0,Y 552.088,Z 134.712,A -85,B 0,C 180,E1 -3093.75,E2 -3093.75} C_VEL
LIN {X 0,Y 552.101,Z 134.711,A -85,B 0,C 180,E1 -3096.748,E2 -3096.748} C_VEL
LIN {X 0,Y 552.146,Z 134.774,A -85,B 0,C 180,E1 -3098.061,E2 -3098.061} C_VEL
LIN {X 0,Y 552.553,Z 140.679,A -85,B 0,C 180,E1 -3099.116,E2 -3099.116} C_VEL
LIN {X 0,Y 552.378,Z 156.487,A -85,B 0,C 180,E1 -3101.911,E2 -3101.911} C_VEL
LIN {X 0,Y 552.22,Z 166.33,A -85,B 0,C 180,E1 -3103.681,E2 -3103.681} C_VEL
LIN {X 0,Y 553.419,Z 174.554,A -85,B 0,C 180,E1 -3103.828,E2 -3103.828} C_VEL
LIN {X 0,Y 553.123,Z 273.964,A -85,B 0,C 180,E1 -3105.146,E2 -3105.146} C_VEL
LIN {X 0,Y 552.999,Z 287.491,A -85,B 0,C 180,E1 -3105.486,E2 -3105.486} C_VEL
LIN {X 0,Y 552.817,Z 300.555,A -85,B 0,C 180,E1 -3105.978,E2 -3105.978} C_VEL
LIN {X 0,Y 552.591,Z 313.048,A -85,B 0,C 180,E1 -3106.623,E2 -3106.623} C_VEL
LIN {X 0,Y 552.44,Z 324.096,A -85,B 0,C 180,E1 -3107.357,E2 -3107.357} C_VEL
LIN {X 0,Y 552.267,Z 334.27,A -85,B 0,C 180,E1 -3108.201,E2 -3108.201} C_VEL
LIN {X 0,Y 552.058,Z 343.574,A -85,B 0,C 180,E1 -3109.153,E2 -3109.153} C_VEL
LIN {X 0,Y 551.971,Z 352.071,A -85,B 0,C 180,E1 -3110.224,E2 -3110.224} C_VEL
LIN {X 0,Y 551.825,Z 359.464,A -85,B 0,C 180,E1 -3111.386,E2 -3111.386} C_VEL
LIN {X 0,Y 551.801,Z 365.272,A -85,B 0,C 180,E1 -3112.543,E2 -3112.543} C_VEL
LIN {X 0,Y 551.774,Z 369.978,A -85,B 0,C 180,E1 -3113.751,E2 -3113.751} C_VEL
LIN {X 0,Y 551.68,Z 373.566,A -85,B 0,C 180,E1 -3115.021,E2 -3115.021} C_VEL
LIN {X 0,Y 551.678,Z 375.276,A -85,B 0,C 180,E1 -3115.907,E2 -3115.907} C_VEL
LIN {X 0,Y 551.67,Z 376.727,A -85,B 0,C 180,E1 -3117.226,E2 -3117.226} C_VEL
LIN {X 0,Y 551.651,Z 376.883,A -85,B 0,C 180,E1 -3118.603,E2 -3118.603} C_VEL
LIN {X 0,Y 551.686,Z 375.513,A -85,B 0,C 180,E1 -3120.027,E2 -3120.027} C_VEL
LIN {X 0,Y 551.707,Z 372.463,A -85,B 0,C 180,E1 -3121.518,E2 -3121.518} C_VEL
LIN {X 0,Y 551.749,Z 368.716,A -85,B 0,C 180,E1 -3122.706,E2 -3122.706} C_VEL
LIN {X 0,Y 551.814,Z 363.476,A -85,B 0,C 180,E1 -3123.934,E2 -3123.934} C_VEL
LIN {X 0,Y 551.869,Z 356.82,A -85,B 0,C 180,E1 -3125.149,E2 -3125.149} C_VEL
LIN {X 0,Y 551.972,Z 349.379,A -85,B 0,C 180,E1 -3126.234,E2 -3126.234} C_VEL
LIN {X 0,Y 552.121,Z 341.63,A -85,B 0,C 180,E1 -3127.155,E2 -3127.155} C_VEL
LIN {X 0,Y 552.297,Z 332.36,A -85,B 0,C 180,E1 -3128.06,E2 -3128.06} C_VEL
LIN {X 0,Y 552.446,Z 321.253,A -85,B 0,C 180,E1 -3128.937,E2 -3128.937} C_VEL
LIN {X 0,Y 552.672,Z 310.26,A -85,B 0,C 180,E1 -3129.628,E2 -3129.628} C_VEL
LIN {X 0,Y 552.799,Z 298.851,A -85,B 0,C 180,E1 -3130.187,E2 -3130.187} C_VEL
LIN {X 0,Y 553,Z 285.304,A -85,B 0,C 180,E1 -3130.671,E2 -3130.671} C_VEL
LIN {X 0,Y 553.139,Z 272.331,A -85,B 0,C 180,E1 -3130.975,E2 -3130.975} C_VEL
LIN {X 0,Y 553.353,Z 173.158,A -85,B 0,C 180,E1 -3132.281,E2 -3132.281} C_VEL
LIN {X 0,Y 552.228,Z 166.369,A -85,B 0,C 180,E1 -3132.406,E2 -3132.406} C_VEL
LIN {X 0,Y 552.462,Z 149.54,A -85,B 0,C 180,E1 -3135.449,E2 -3135.449} C_VEL
LIN {X 0,Y 552.539,Z 137.105,A -85,B 0,C 180,E1 -3137.699,E2 -3137.699} C_VEL
LIN {X 0,Y 552.171,Z 134.707,A -85,B 0,C 180,E1 -3138.156,E2 -3138.156} C_VEL
LIN {X 0,Y 552.138,Z 134.706,A -85,B 0,C 180,E1 -3141.214,E2 -3141.214} C_VEL
LIN {X 0,Y 552.189,Z 134.702,A -85,B 0,C 180,E1 -3144.156,E2 -3144.156} C_VEL
LIN {X 0,Y 552.224,Z 134.694,A -85,B 0,C 180,E1 -3147.812,E2 -3147.812} C_VEL
LIN {X 0,Y 552.236,Z 134.695,A -85,B 0,C 180,E1 -3150.729,E2 -3150.729} C_VEL
LIN {X 0,Y 552.187,Z 134.698,A -85,B 0,C 180,E1 -3152.918,E2 -3152.918} C_VEL
LIN {X 0,Y 552.188,Z 134.7,A -85,B 0,C 180,E1 -3155.844,E2 -3155.844} C_VEL
LIN {X 0,Y 552.137,Z 134.704,A -85,B 0,C 180,E1 -3158.786,E2 -3158.786} C_VEL
LIN {X 0,Y 552.16,Z 134.704,A -85,B 0,C 180,E1 -3161.751,E2 -3161.751} C_VEL
LIN {X 0,Y 552.131,Z 134.704,A -85,B 0,C 180,E1 -3164.749,E2 -3164.749} C_VEL
LIN {X 0,Y 552.082,Z 134.717,A -85,B 0,C 180,E1 -3167.79,E2 -3167.79} C_VEL
LIN {X 0,Y 552.122,Z 134.711,A -85,B 0,C 180,E1 -3170.102,E2 -3170.102} C_VEL
LIN {X 0,Y 552.086,Z 134.711,A -85,B 0,C 180,E1 -3172.451,E2 -3172.451} C_VEL
LIN {X 0,Y 552.086,Z 134.713,A -85,B 0,C 180,E1 -3175.334,E2 -3175.334} C_VEL
LIN {X 0,Y 552.06,Z 134.716,A -85,B 0,C 180,E1 -3178.101,E2 -3178.101} C_VEL
LIN {X 0,Y 552.095,Z 134.708,A -85,B 0,C 180,E1 -3180.61,E2 -3180.61} C_VEL
LIN {X 0,Y 552.107,Z 134.71,A -85,B 0,C 180,E1 -3183.187,E2 -3183.187} C_VEL
LIN {X 0,Y 552.073,Z 134.715,A -85,B 0,C 180,E1 -3185.845,E2 -3185.845} C_VEL
LIN {X 0,Y 552.115,Z 134.706,A -85,B 0,C 180,E1 -3188.59,E2 -3188.59} C_VEL
LIN {X 0,Y 552.076,Z 134.719,A -85,B 0,C 180,E1 -3191.45,E2 -3191.45} C_VEL
LIN {X 0,Y 552.078,Z 134.711,A -85,B 0,C 180,E1 -3194.53,E2 -3194.53} C_VEL
LIN {X 0,Y 552.089,Z 134.713,A -85,B 0,C 180,E1 -3197.59,E2 -3197.59} C_VEL
LIN {X 0,Y 552.128,Z 134.705,A -85,B 0,C 180,E1 -3200.472,E2 -3200.472} C_VEL
LIN {X 0,Y 552.102,Z 134.713,A -85,B 0,C 180,E1 -3203.318,E2 -3203.318} C_VEL
LIN {X 0,Y 552.101,Z 134.708,A -85,B 0,C 180,E1 -3205.937,E2 -3205.937} C_VEL
LIN {X 0,Y 552.083,Z 134.713,A -85,B 0,C 180,E1 -3208.538,E2 -3208.538} C_VEL
LIN {X 0,Y 552.081,Z 134.712,A -85,B 0,C 180,E1 -3211.447,E2 -3211.447} C_VEL
LIN {X 0,Y 552.085,Z 134.712,A -85,B 0,C 180,E1 -3214.353,E2 -3214.353} C_VEL
LIN {X 0,Y 552.071,Z 134.721,A -85,B 0,C 180,E1 -3216.757,E2 -3216.757} C_VEL
LIN {X 0,Y 552.1,Z 134.711,A -85,B 0,C 180,E1 -3219.119,E2 -3219.119} C_VEL
LIN {X 0,Y 552.082,Z 134.71,A -85,B 0,C 180,E1 -3221.443,E2 -3221.443} C_VEL
LIN {X 0,Y 552.088,Z 134.718,A -85,B 0,C 180,E1 -3224.495,E2 -3224.495} C_VEL
LIN {X 0,Y 552.1,Z 134.708,A -85,B 0,C 180,E1 -3227.502,E2 -3227.502} C_VEL
LIN {X 0,Y 552.098,Z 134.709,A -85,B 0,C 180,E1 -3229.734,E2 -3229.734} C_VEL
LIN {X 0,Y 552.113,Z 134.709,A -85,B 0,C 180,E1 -3231.951,E2 -3231.951} C_VEL
LIN {X 0,Y 552.207,Z 134.696,A -85,B 0,C 180,E1 -3234.889,E2 -3234.889} C_VEL
LIN {X 0,Y 552.222,Z 134.696,A -85,B 0,C 180,E1 -3237.812,E2 -3237.812} C_VEL
LIN {X 0,Y 552.226,Z 134.698,A -85,B 0,C 180,E1 -3240,E2 -3240} C_VEL
LIN {X 0,Y 552.179,Z 134.698,A -85,B 0,C 180,E1 -3242.918,E2 -3242.918} C_VEL
LIN {X 0,Y 552.176,Z 134.704,A -85,B 0,C 180,E1 -3245.844,E2 -3245.844} C_VEL
LIN {X 0,Y 552.127,Z 134.705,A -85,B 0,C 180,E1 -3248.786,E2 -3248.786} C_VEL
LIN {X 0,Y 552.102,Z 134.715,A -85,B 0,C 180,E1 -3251.752,E2 -3251.752} C_VEL
LIN {X 0,Y 552.093,Z 134.708,A -85,B 0,C 180,E1 -3254.75,E2 -3254.75} C_VEL
LIN {X 0,Y 552.073,Z 134.72,A -85,B 0,C 180,E1 -3257.79,E2 -3257.79} C_VEL
LIN {X 0,Y 552.051,Z 134.717,A -85,B 0,C 180,E1 -3260.104,E2 -3260.104} C_VEL
LIN {X 0,Y 552.044,Z 134.715,A -85,B 0,C 180,E1 -3262.453,E2 -3262.453} C_VEL
LIN {X 0,Y 552.076,Z 134.716,A -85,B 0,C 180,E1 -3265.331,E2 -3265.331} C_VEL
LIN {X 0,Y 552.051,Z 134.715,A -85,B 0,C 180,E1 -3268.102,E2 -3268.102} C_VEL
LIN {X 0,Y 552.07,Z 134.712,A -85,B 0,C 180,E1 -3270.611,E2 -3270.611} C_VEL
LIN {X 0,Y 552.092,Z 134.715,A -85,B 0,C 180,E1 -3273.188,E2 -3273.188} C_VEL
LIN {X 0,Y 552.068,Z 134.714,A -85,B 0,C 180,E1 -3275.845,E2 -3275.845} C_VEL
LIN {X 0,Y 552.087,Z 134.71,A -85,B 0,C 180,E1 -3278.592,E2 -3278.592} C_VEL
LIN {X 0,Y 552.058,Z 134.718,A -85,B 0,C 180,E1 -3281.452,E2 -3281.452} C_VEL
LIN {X 0,Y 552.073,Z 134.713,A -85,B 0,C 180,E1 -3284.529,E2 -3284.529} C_VEL
LIN {X 0,Y 552.082,Z 134.712,A -85,B 0,C 180,E1 -3287.59,E2 -3287.59} C_VEL
LIN {X 0,Y 552.083,Z 134.712,A -85,B 0,C 180,E1 -3290.468,E2 -3290.468} C_VEL
LIN {X 0,Y 552.052,Z 134.717,A -85,B 0,C 180,E1 -3293.325,E2 -3293.325} C_VEL
LIN {X 0,Y 552.084,Z 134.71,A -85,B 0,C 180,E1 -3295.936,E2 -3295.936} C_VEL
LIN {X 0,Y 552.081,Z 134.716,A -85,B 0,C 180,E1 -3298.538,E2 -3298.538} C_VEL
LIN {X 0,Y 552.071,Z 134.713,A -85,B 0,C 180,E1 -3301.449,E2 -3301.449} C_VEL
LIN {X 0,Y 552.062,Z 134.72,A -85,B 0,C 180,E1 -3304.352,E2 -3304.352} C_VEL
LIN {X 0,Y 552.095,Z 134.841,A -85,B 0,C 180,E1 -3306.547,E2 -3306.547} C_VEL
LIN {X 0,Y 553.066,Z 141.282,A -85,B 0,C 180,E1 -3307.591,E2 -3307.591} C_VEL
LIN {X 0,Y 552.8,Z 159.957,A -85,B 0,C 180,E1 -3310.442,E2 -3310.442} C_VEL
LIN {X 0,Y 552.519,Z 179.45,A -85,B 0,C 180,E1 -3313.369,E2 -3313.369} C_VEL
LIN {X 0,Y 552.353,Z 194.648,A -85,B 0,C 180,E1 -3315.628,E2 -3315.628} C_VEL
LIN {X 0,Y 553.4,Z 202.493,A -85,B 0,C 180,E1 -3315.764,E2 -3315.764} C_VEL
LIN {X 0,Y 553.137,Z 302.641,A -85,B 0,C 180,E1 -3317.083,E2 -3317.083} C_VEL
LIN {X 0,Y 552.981,Z 315.97,A -85,B 0,C 180,E1 -3317.406,E2 -3317.406} C_VEL
LIN {X 0,Y 552.847,Z 328.168,A -85,B 0,C 180,E1 -3317.845,E2 -3317.845} C_VEL
LIN {X 0,Y 552.654,Z 339.023,A -85,B 0,C 180,E1 -3318.366,E2 -3318.366} C_VEL
LIN {X 0,Y 552.479,Z 350.786,A -85,B 0,C 180,E1 -3319.092,E2 -3319.092} C_VEL
LIN {X 0,Y 552.297,Z 361.464,A -85,B 0,C 180,E1 -3319.923,E2 -3319.923} C_VEL
LIN {X 0,Y 552.126,Z 371.083,A -85,B 0,C 180,E1 -3320.845,E2 -3320.845} C_VEL
LIN {X 0,Y 552.013,Z 378.96,A -85,B 0,C 180,E1 -3321.765,E2 -3321.765} C_VEL
LIN {X 0,Y 551.889,Z 386.621,A -85,B 0,C 180,E1 -3322.868,E2 -3322.868} C_VEL
LIN {X 0,Y 551.867,Z 393.679,A -85,B 0,C 180,E1 -3324.153,E2 -3324.153} C_VEL
LIN {X 0,Y 551.725,Z 398.373,A -85,B 0,C 180,E1 -3325.251,E2 -3325.251} C_VEL
LIN {X 0,Y 551.75,Z 401.958,A -85,B 0,C 180,E1 -3326.348,E2 -3326.348} C_VEL
LIN {X 0,Y 551.723,Z 403.807,A -85,B 0,C 180,E1 -3327.079,E2 -3327.079} C_VEL
LIN {X 0,Y 551.645,Z 406.182,A -85,B 0,C 180,E1 -3328.54,E2 -3328.54} C_VEL
LIN {X 0,Y 551.64,Z 407,A -85,B 0,C 180,E1 -3330,E2 -3330} C_VEL
LIN {X 0,Y 551.645,Z 406.183,A -85,B 0,C 180,E1 -3331.46,E2 -3331.46} C_VEL
LIN {X 0,Y 551.723,Z 403.81,A -85,B 0,C 180,E1 -3332.921,E2 -3332.921} C_VEL
LIN {X 0,Y 551.764,Z 400.895,A -85,B 0,C 180,E1 -3334.017,E2 -3334.017} C_VEL
LIN {X 0,Y 551.723,Z 396.948,A -85,B 0,C 180,E1 -3335.116,E2 -3335.116} C_VEL
LIN {X 0,Y 551.803,Z 391.188,A -85,B 0,C 180,E1 -3336.342,E2 -3336.342} C_VEL
LIN {X 0,Y 551.926,Z 384.234,A -85,B 0,C 180,E1 -3337.5,E2 -3337.5} C_VEL
LIN {X 0,Y 552.082,Z 375.986,A -85,B 0,C 180,E1 -3338.603,E2 -3338.603} C_VEL
LIN {X 0,Y 552.2,Z 367.492,A -85,B 0,C 180,E1 -3339.524,E2 -3339.524} C_VEL
LIN {X 0,Y 552.429,Z 356.996,A -85,B 0,C 180,E1 -3340.445,E2 -3340.445} C_VEL
LIN {X 0,Y 552.575,Z 346.144,A -85,B 0,C 180,E1 -3341.214,E2 -3341.214} C_VEL
LIN {X 0,Y 552.752,Z 335.219,A -85,B 0,C 180,E1 -3341.831,E2 -3341.831} C_VEL
LIN {X 0,Y 552.899,Z 323.525,A -85,B 0,C 180,E1 -3342.34,E2 -3342.34} C_VEL
LIN {X 0,Y 553.039,Z 310.963,A -85,B 0,C 180,E1 -3342.733,E2 -3342.733} C_VEL
LIN {X 0,Y 553.163,Z 298.22,A -85,B 0,C 180,E1 -3342.987,E2 -3342.987} C_VEL
LIN {X 0,Y 553.221,Z 200.469,A -85,B 0,C 180,E1 -3344.266,E2 -3344.266} C_VEL
LIN {X 0,Y 552.333,Z 194.438,A -85,B 0,C 180,E1 -3344.393,E2 -3344.393} C_VEL
LIN {X 0,Y 552.543,Z 174.589,A -85,B 0,C 180,E1 -3347.337,E2 -3347.337} C_VEL
LIN {X 0,Y 552.825,Z 156.34,A -85,B 0,C 180,E1 -3350.075,E2 -3350.075} C_VEL
LIN {X 0,Y 553.014,Z 140.963,A -85,B 0,C 180,E1 -3352.412,E2 -3352.412} C_VEL
LIN {X 0,Y 552.072,Z 134.721,A -85,B 0,C 180,E1 -3353.424,E2 -3353.424} C_VEL
LIN {X 0,Y 552.07,Z 134.713,A -85,B 0,C 180,E1 -3356.459,E2 -3356.459} C_VEL
LIN {X 0,Y 552.037,Z 134.721,A -85,B 0,C 180,E1 -3358.933,E2 -3358.933} C_VEL
LIN {X 0,Y 552.094,Z 134.717,A -85,B 0,C 180,E1 -3361.472,E2 -3361.472} C_VEL
LIN {X 0,Y 552.072,Z 134.713,A -85,B 0,C 180,E1 -3364.161,E2 -3364.161} C_VEL
LIN {X 0,Y 552.047,Z 134.718,A -85,B 0,C 180,E1 -3366.752,E2 -3366.752} C_VEL
LIN {X 0,Y 552.072,Z 134.715,A -85,B 0,C 180,E1 -3369.533,E2 -3369.533} C_VEL
LIN {X 0,Y 552.081,Z 134.712,A -85,B 0,C 180,E1 -3372.431,E2 -3372.431} C_VEL
LIN {X 0,Y 552.069,Z 134.714,A -85,B 0,C 180,E1 -3375.56,E2 -3375.56} C_VEL
LIN {X 0,Y 552.054,Z 134.717,A -85,B 0,C 180,E1 -3378.548,E2 -3378.548} C_VEL
LIN {X 0,Y 552.074,Z 134.714,A -85,B 0,C 180,E1 -3381.407,E2 -3381.407} C_VEL
LIN {X 0,Y 552.056,Z 134.718,A -85,B 0,C 180,E1 -3384.564,E2 -3384.564} C_VEL
LIN {X 0,Y 552.091,Z 134.712,A -85,B 0,C 180,E1 -3387.158,E2 -3387.158} C_VEL
LIN {X 0,Y 552.069,Z 134.712,A -85,B 0,C 180,E1 -3389.959,E2 -3389.959} C_VEL
LIN {X 0,Y 552.079,Z 134.714,A -85,B 0,C 180,E1 -3393.013,E2 -3393.013} C_VEL
LIN {X 0,Y 552.065,Z 134.712,A -85,B 0,C 180,E1 -3395.96,E2 -3395.96} C_VEL
LIN {X 0,Y 552.069,Z 134.711,A -85,B 0,C 180,E1 -3399.118,E2 -3399.118} C_VEL
LIN {X 0,Y 552.048,Z 134.714,A -85,B 0,C 180,E1 -3401.442,E2 -3401.442} C_VEL
LIN {X 0,Y 552.074,Z 134.711,A -85,B 0,C 180,E1 -3403.736,E2 -3403.736} C_VEL
LIN {X 0,Y 552.087,Z 134.713,A -85,B 0,C 180,E1 -3406.754,E2 -3406.754} C_VEL
LIN {X 0,Y 552.129,Z 134.704,A -85,B 0,C 180,E1 -3408.993,E2 -3408.993} C_VEL
LIN {X 0,Y 552.111,Z 134.71,A -85,B 0,C 180,E1 -3411.951,E2 -3411.951} C_VEL
LIN {X 0,Y 552.204,Z 134.696,A -85,B 0,C 180,E1 -3414.889,E2 -3414.889} C_VEL
LIN {X 0,Y 552.221,Z 134.695,A -85,B 0,C 180,E1 -3417.812,E2 -3417.812} C_VEL
LIN {X 0,Y 552.226,Z 134.699,A -85,B 0,C 180,E1 -3420,E2 -3420} C_VEL
LIN {X 0,Y 552.177,Z 134.698,A -85,B 0,C 180,E1 -3422.918,E2 -3422.918} C_VEL
LIN {X 0,Y 552.176,Z 134.704,A -85,B 0,C 180,E1 -3425.844,E2 -3425.844} C_VEL
LIN {X 0,Y 552.128,Z 134.704,A -85,B 0,C 180,E1 -3428.786,E2 -3428.786} C_VEL
LIN {X 0,Y 552.105,Z 134.714,A -85,B 0,C 180,E1 -3431.752,E2 -3431.752} C_VEL
LIN {X 0,Y 552.124,Z 134.705,A -85,B 0,C 180,E1 -3434.749,E2 -3434.749} C_VEL
LIN {X 0,Y 552.077,Z 134.72,A -85,B 0,C 180,E1 -3437.79,E2 -3437.79} C_VEL
LIN {X 0,Y 552.095,Z 134.713,A -85,B 0,C 180,E1 -3440.103,E2 -3440.103} C_VEL
LIN {X 0,Y 552.048,Z 134.715,A -85,B 0,C 180,E1 -3442.453,E2 -3442.453} C_VEL
LIN {X 0,Y 552.087,Z 134.715,A -85,B 0,C 180,E1 -3445.334,E2 -3445.334} C_VEL
LIN {X 0,Y 552.053,Z 134.717,A -85,B 0,C 180,E1 -3448.102,E2 -3448.102} C_VEL
LIN {X 0,Y 552.075,Z 134.712,A -85,B 0,C 180,E1 -3450.611,E2 -3450.611} C_VEL
LIN {X 0,Y 552.108,Z 134.713,A -85,B 0,C 180,E1 -3453.187,E2 -3453.187} C_VEL
LIN {X 0,Y 552.088,Z 134.712,A -85,B 0,C 180,E1 -3453.75,E2 -3453.75} C_VEL
LIN {X 0,Y 551.444,Z 134.794,A -85,B 0,C 180,E1 -3454.359,E2 -3454.359} C_VEL
LIN {X 0,Y 548.627,Z 135.15,A -85,B 0,C 180,E1 -3455.347,E2 -3455.347} C_VEL
LIN {X 0,Y 546.221,Z 135.446,A -85,B 0,C 180,E1 -3456.143,E2 -3456.143} C_VEL
LIN {X 0,Y 545.164,Z 135.576,A -85,B 0,C 180,E1 -3456.757,E2 -3456.757} C_VEL
LIN {X 0,Y 545.066,Z 135.59,A -85,B 0,C 180,E1 -3456.965,E2 -3456.965} C_VEL
LIN {X 0,Y 545.102,Z 135.612,A -85,B 0,C 180,E1 -3457.956,E2 -3457.956} C_VEL
LIN {X 0,Y 545.535,Z 140.861,A -85,B 0,C 180,E1 -3458.906,E2 -3458.906} C_VEL
LIN {X 0,Y 545.378,Z 157.236,A -85,B 0,C 180,E1 -3461.822,E2 -3461.822} C_VEL
LIN {X 0,Y 545.229,Z 166.526,A -85,B 0,C 180,E1 -3463.491,E2 -3463.491} C_VEL
LIN {X 0,Y 546.54,Z 174.795,A -85,B 0,C 180,E1 -3463.647,E2 -3463.647} C_VEL
LIN {X 0,Y 546.199,Z 273.978,A -85,B 0,C 180,E1 -3464.979,E2 -3464.979} C_VEL
LIN {X 0,Y 546.105,Z 287.197,A -85,B 0,C 180,E1 -3465.312,E2 -3465.312} C_VEL
LIN {X 0,Y 545.929,Z 299.423,A -85,B 0,C 180,E1 -3465.766,E2 -3465.766} C_VEL
LIN {X 0,Y 545.712,Z 311.449,A -85,B 0,C 180,E1 -3466.373,E2 -3466.373} C_VEL
LIN {X 0,Y 545.467,Z 323.064,A -85,B 0,C 180,E1 -3467.131,E2 -3467.131} C_VEL
LIN {X 0,Y 545.307,Z 332.74,A -85,B 0,C 180,E1 -3467.918,E2 -3467.918} C_VEL
LIN {X 0,Y 545.07,Z 342.415,A -85,B 0,C 180,E1 -3468.884,E2 -3468.884} C_VEL
LIN {X 0,Y 544.938,Z 350.259,A -85,B 0,C 180,E1 -3469.846,E2 -3469.846} C_VEL
LIN {X 0,Y 544.811,Z 358.11,A -85,B 0,C 180,E1 -3471.033,E2 -3471.033} C_VEL
LIN {X 0,Y 544.724,Z 364.664,A -85,B 0,C 180,E1 -3472.289,E2 -3472.289} C_VEL
LIN {X 0,Y 544.673,Z 369.785,A -85,B 0,C 180,E1 -3473.591,E2 -3473.591} C_VEL
LIN {X 0,Y 544.598,Z 373.629,A -85,B 0,C 180,E1 -3474.951,E2 -3474.951} C_VEL
LIN {X 0,Y 544.557,Z 376.009,A -85,B 0,C 180,E1 -3476.292,E2 -3476.292} C_VEL
LIN {X 0,Y 544.569,Z 376.82,A -85,B 0,C 180,E1 -3477.177,E2 -3477.177} C_VEL
LIN {X 0,Y 544.545,Z 377.044,A -85,B 0,C 180,E1 -3478.409,E2 -3478.409} C_VEL
LIN {X 0,Y 544.598,Z 375.951,A -85,B 0,C 180,E1 -3479.841,E2 -3479.841} C_VEL
LIN {X 0,Y 544.588,Z 374.667,A -85,B 0,C 180,E1 -3480.633,E2 -3480.633} C_VEL
LIN {X 0,Y 544.618,Z 371.656,A -85,B 0,C 180,E1 -3481.9,E2 -3481.9} C_VEL
LIN {X 0,Y 544.67,Z 367.4,A -85,B 0,C 180,E1 -3483.152,E2 -3483.152} C_VEL
LIN {X 0,Y 544.774,Z 362.218,A -85,B 0,C 180,E1 -3484.307,E2 -3484.307} C_VEL
LIN {X 0,Y 544.854,Z 355.924,A -85,B 0,C 180,E1 -3485.418,E2 -3485.418} C_VEL
LIN {X 0,Y 544.944,Z 348.823,A -85,B 0,C 180,E1 -3486.434,E2 -3486.434} C_VEL
LIN {X 0,Y 545.108,Z 340.171,A -85,B 0,C 180,E1 -3487.445,E2 -3487.445} C_VEL
LIN {X 0,Y 545.325,Z 330.908,A -85,B 0,C 180,E1 -3488.331,E2 -3488.331} C_VEL
LIN {X 0,Y 545.497,Z 320.41,A -85,B 0,C 180,E1 -3489.15,E2 -3489.15} C_VEL
LIN {X 0,Y 545.754,Z 309.221,A -85,B 0,C 180,E1 -3489.841,E2 -3489.841} C_VEL
LIN {X 0,Y 545.909,Z 296.545,A -85,B 0,C 180,E1 -3490.444,E2 -3490.444} C_VEL
LIN {X 0,Y 546.123,Z 283.417,A -85,B 0,C 180,E1 -3490.892,E2 -3490.892} C_VEL
LIN {X 0,Y 546.223,Z 270.989,A -85,B 0,C 180,E1 -3491.163,E2 -3491.163} C_VEL
LIN {X 0,Y 546.545,Z 174.196,A -85,B 0,C 180,E1 -3492.45,E2 -3492.45} C_VEL
LIN {X 0,Y 545.255,Z 166.548,A -85,B 0,C 180,E1 -3492.595,E2 -3492.595} C_VEL
LIN {X 0,Y 545.478,Z 150.76,A -85,B 0,C 180,E1 -3495.468,E2 -3495.468} C_VEL
LIN {X 0,Y 545.566,Z 138.395,A -85,B 0,C 180,E1 -3497.728,E2 -3497.728} C_VEL
LIN {X 0,Y 545.153,Z 135.582,A -85,B 0,C 180,E1 -3498.294,E2 -3498.294} C_VEL
LIN {X 0,Y 545.099,Z 135.584,A -85,B 0,C 180,E1 -3501.1,E2 -3501.1} C_VEL
LIN {X 0,Y 545.139,Z 135.579,A -85,B 0,C 180,E1 -3504.08,E2 -3504.08} C_VEL
LIN {X 0,Y 545.161,Z 135.574,A -85,B 0,C 180,E1 -3507.044,E2 -3507.044} C_VEL
LIN {X 0,Y 545.197,Z 135.571,A -85,B 0,C 180,E1 -3510,E2 -3510} C_VEL
LIN {X 0,Y 545.154,Z 135.574,A -85,B 0,C 180,E1 -3512.956,E2 -3512.956} C_VEL
LIN {X 0,Y 545.137,Z 135.58,A -85,B 0,C 180,E1 -3515.92,E2 -3515.92} C_VEL
LIN {X 0,Y 545.098,Z 135.581,A -85,B 0,C 180,E1 -3518.9,E2 -3518.9} C_VEL
LIN {X 0,Y 545.103,Z 135.586,A -85,B 0,C 180,E1 -3521.905,E2 -3521.905} C_VEL
LIN {X 0,Y 545.083,Z 135.582,A -85,B 0,C 180,E1 -3524.944,E2 -3524.944} C_VEL
LIN {X 0,Y 545.051,Z 135.594,A -85,B 0,C 180,E1 -3528.027,E2 -3528.027} C_VEL
LIN {X 0,Y 545.087,Z 135.584,A -85,B 0,C 180,E1 -3530.373,E2 -3530.373} C_VEL
LIN {X 0,Y 545.074,Z 135.588,A -85,B 0,C 180,E1 -3533.56,E2 -3533.56} C_VEL
LIN {X 0,Y 545.058,Z 135.585,A -85,B 0,C 180,E1 -3536.827,E2 -3536.827} C_VEL
LIN {X 0,Y 545.029,Z 135.593,A -85,B 0,C 180,E1 -3539.341,E2 -3539.341} C_VEL
LIN {X 0,Y 545.055,Z 135.59,A -85,B 0,C 180,E1 -3541.915,E2 -3541.915} C_VEL
LIN {X 0,Y 545.049,Z 135.586,A -85,B 0,C 180,E1 -3544.566,E2 -3544.566} C_VEL
LIN {X 0,Y 545.032,Z 135.595,A -85,B 0,C 180,E1 -3547.305,E2 -3547.305} C_VEL
LIN {X 0,Y 545.065,Z 135.585,A -85,B 0,C 180,E1 -3550.143,E2 -3550.143} C_VEL
LIN {X 0,Y 545.02,Z 135.596,A -85,B 0,C 180,E1 -3553.113,E2 -3553.113} C_VEL
LIN {X 0,Y 545.031,Z 135.588,A -85,B 0,C 180,E1 -3556.229,E2 -3556.229} C_VEL
LIN {X 0,Y 545.031,Z 135.593,A -85,B 0,C 180,E1 -3558.88,E2 -3558.88} C_VEL
LIN {X 0,Y 545.05,Z 135.587,A -85,B 0,C 180,E1 -3561.762,E2 -3561.762} C_VEL
LIN {X 0,Y 545.028,Z 135.591,A -85,B 0,C 180,E1 -3564.531,E2 -3564.531} C_VEL
LIN {X 0,Y 545.065,Z 135.59,A -85,B 0,C 180,E1 -3567.211,E2 -3567.211} C_VEL
LIN {X 0,Y 545.03,Z 135.588,A -85,B 0,C 180,E1 -3569.808,E2 -3569.808} C_VEL
LIN {X 0,Y 545.039,Z 135.597,A -85,B 0,C 180,E1 -3572.839,E2 -3572.839} C_VEL
LIN {X 0,Y 545.019,Z 135.59,A -85,B 0,C 180,E1 -3575.629,E2 -3575.629} C_VEL
LIN {X 0,Y 545.039,Z 135.595,A -85,B 0,C 180,E1 -3578.835,E2 -3578.835} C_VEL
LIN {X 0,Y 545.045,Z 135.588,A -85,B 0,C 180,E1 -3581.194,E2 -3581.194} C_VEL
LIN {X 0,Y 545.035,Z 135.593,A -85,B 0,C 180,E1 -3584.289,E2 -3584.289} C_VEL
LIN {X 0,Y 545.041,Z 135.596,A -85,B 0,C 180,E1 -3586.579,E2 -3586.579} C_VEL
LIN {X 0,Y 545.12,Z 135.581,A -85,B 0,C 180,E1 -3588.849,E2 -3588.849} C_VEL
LIN {X 0,Y 545.07,Z 135.585,A -85,B 0,C 180,E1 -3591.846,E2 -3591.846} C_VEL
LIN {X 0,Y 545.165,Z 135.574,A -85,B 0,C 180,E1 -3594.823,E2 -3594.823} C_VEL
LIN {X 0,Y 545.193,Z 135.571,A -85,B 0,C 180,E1 -3597.784,E2 -3597.784} C_VEL
LIN {X 0,Y 545.195,Z 135.574,A -85,B 0,C 180,E1 -3600,E2 -3600} C_VEL
LIN {X 0,Y 545.146,Z 135.574,A -85,B 0,C 180,E1 -3602.956,E2 -3602.956} C_VEL
LIN {X 0,Y 545.127,Z 135.584,A -85,B 0,C 180,E1 -3605.92,E2 -3605.92} C_VEL
LIN {X 0,Y 545.071,Z 135.583,A -85,B 0,C 180,E1 -3608.901,E2 -3608.901} C_VEL
LIN {X 0,Y 545.067,Z 135.593,A -85,B 0,C 180,E1 -3611.906,E2 -3611.906} C_VEL
LIN {X 0,Y 545.043,Z 135.587,A -85,B 0,C 180,E1 -3614.945,E2 -3614.945} C_VEL
LIN {X 0,Y 545.037,Z 135.593,A -85,B 0,C 180,E1 -3618.027,E2 -3618.027} C_VEL
LIN {X 0,Y 545.007,Z 135.592,A -85,B 0,C 180,E1 -3620.376,E2 -3620.376} C_VEL
LIN {X 0,Y 544.99,Z 135.593,A -85,B 0,C 180,E1 -3622.76,E2 -3622.76} C_VEL
LIN {X 0,Y 545.028,Z 135.597,A -85,B 0,C 180,E1 -3625.493,E2 -3625.493} C_VEL
LIN {X 0,Y 545.035,Z 135.588,A -85,B 0,C 180,E1 -3628.496,E2 -3628.496} C_VEL
LIN {X 0,Y 545.046,Z 135.592,A -85,B 0,C 180,E1 -3631.676,E2 -3631.676} C_VEL
LIN {X 0,Y 545.041,Z 135.587,A -85,B 0,C 180,E1 -3634.566,E2 -3634.566} C_VEL
LIN {X 0,Y 545.008,Z 135.6,A -85,B 0,C 180,E1 -3637.306,E2 -3637.306} C_VEL
LIN {X 0,Y 545.034,Z 135.588,A -85,B 0,C 180,E1 -3640.146,E2 -3640.146} C_VEL
LIN {X 0,Y 545.019,Z 135.599,A -85,B 0,C 180,E1 -3643.113,E2 -3643.113} C_VEL
LIN {X 0,Y 545.027,Z 135.589,A -85,B 0,C 180,E1 -3646.229,E2 -3646.229} C_VEL
LIN {X 0,Y 545.006,Z 135.599,A -85,B 0,C 180,E1 -3648.878,E2 -3648.878} C_VEL
LIN {X 0,Y 545.026,Z 135.589,A -85,B 0,C 180,E1 -3651.867,E2 -3651.867} C_VEL
LIN {X 0,Y 545.018,Z 135.594,A -85,B 0,C 180,E1 -3654.53,E2 -3654.53} C_VEL
LIN {X 0,Y 545.051,Z 135.589,A -85,B 0,C 180,E1 -3657.21,E2 -3657.21} C_VEL
LIN {X 0,Y 545.018,Z 135.591,A -85,B 0,C 180,E1 -3659.807,E2 -3659.807} C_VEL
LIN {X 0,Y 544.998,Z 135.598,A -85,B 0,C 180,E1 -3662.339,E2 -3662.339} C_VEL
LIN {X 0,Y 545.023,Z 135.598,A -85,B 0,C 180,E1 -3664.815,E2 -3664.815} C_VEL
LIN {X 0,Y 545.056,Z 135.796,A -85,B 0,C 180,E1 -3666.402,E2 -3666.402} C_VEL
LIN {X 0,Y 546.108,Z 142.301,A -85,B 0,C 180,E1 -3667.474,E2 -3667.474} C_VEL
LIN {X 0,Y 545.841,Z 159.612,A -85,B 0,C 180,E1 -3670.156,E2 -3670.156} C_VEL
LIN {X 0,Y 545.525,Z 178.009,A -85,B 0,C 180,E1 -3672.957,E2 -3672.957} C_VEL
LIN {X 0,Y 545.327,Z 194.502,A -85,B 0,C 180,E1 -3675.445,E2 -3675.445} C_VEL
LIN {X 0,Y 546.515,Z 203.485,A -85,B 0,C 180,E1 -3675.597,E2 -3675.597} C_VEL
LIN {X 0,Y 546.22,Z 302.338,A -85,B 0,C 180,E1 -3676.916,E2 -3676.916} C_VEL
LIN {X 0,Y 546.04,Z 315.706,A -85,B 0,C 180,E1 -3677.243,E2 -3677.243} C_VEL
LIN {X 0,Y 545.872,Z 329.048,A -85,B 0,C 180,E1 -3677.735,E2 -3677.735} C_VEL
LIN {X 0,Y 545.644,Z 340.689,A -85,B 0,C 180,E1 -3678.322,E2 -3678.322} C_VEL
LIN {X 0,Y 545.45,Z 351.86,A -85,B 0,C 180,E1 -3679.044,E2 -3679.044} C_VEL
LIN {X 0,Y 545.26,Z 362.321,A -85,B 0,C 180,E1 -3679.885,E2 -3679.885} C_VEL
LIN {X 0,Y 545.085,Z 370.872,A -85,B 0,C 180,E1 -3680.725,E2 -3680.725} C_VEL
LIN {X 0,Y 544.947,Z 378.76,A -85,B 0,C 180,E1 -3681.658,E2 -3681.658} C_VEL
LIN {X 0,Y 544.824,Z 386.463,A -85,B 0,C 180,E1 -3682.775,E2 -3682.775} C_VEL
LIN {X 0,Y 544.777,Z 393.563,A -85,B 0,C 180,E1 -3684.076,E2 -3684.076} C_VEL
LIN {X 0,Y 544.628,Z 398.281,A -85,B 0,C 180,E1 -3685.188,E2 -3685.188} C_VEL
LIN {X 0,Y 544.669,Z 401.889,A -85,B 0,C 180,E1 -3686.301,E2 -3686.301} C_VEL
LIN {X 0,Y 544.65,Z 403.749,A -85,B 0,C 180,E1 -3687.041,E2 -3687.041} C_VEL
LIN {X 0,Y 544.546,Z 406.137,A -85,B 0,C 180,E1 -3688.521,E2 -3688.521} C_VEL
LIN {X 0,Y 544.542,Z 406.744,A -85,B 0,C 180,E1 -3689.261,E2 -3689.261} C_VEL
LIN {X 0,Y 544.541,Z 406.96,A -85,B 0,C 180,E1 -3690,E2 -3690} C_VEL
LIN {X 0,Y 544.546,Z 406.138,A -85,B 0,C 180,E1 -3691.479,E2 -3691.479} C_VEL
LIN {X 0,Y 544.65,Z 403.752,A -85,B 0,C 180,E1 -3692.959,E2 -3692.959} C_VEL
LIN {X 0,Y 544.684,Z 400.819,A -85,B 0,C 180,E1 -3694.07,E2 -3694.07} C_VEL
LIN {X 0,Y 544.653,Z 396.845,A -85,B 0,C 180,E1 -3695.182,E2 -3695.182} C_VEL
LIN {X 0,Y 544.713,Z 391.568,A -85,B 0,C 180,E1 -3696.328,E2 -3696.328} C_VEL
LIN {X 0,Y 544.836,Z 385.293,A -85,B 0,C 180,E1 -3697.411,E2 -3697.411} C_VEL
LIN {X 0,Y 544.988,Z 377.259,A -85,B 0,C 180,E1 -3698.529,E2 -3698.529} C_VEL
LIN {X 0,Y 545.114,Z 369.069,A -85,B 0,C 180,E1 -3699.461,E2 -3699.461} C_VEL
LIN {X 0,Y 545.365,Z 359.082,A -85,B 0,C 180,E1 -3700.394,E2 -3700.394} C_VEL
LIN {X 0,Y 545.548,Z 348.217,A -85,B 0,C 180,E1 -3701.208,E2 -3701.208} C_VEL
LIN {X 0,Y 545.712,Z 336.738,A -85,B 0,C 180,E1 -3701.892,E2 -3701.892} C_VEL
LIN {X 0,Y 545.93,Z 324.478,A -85,B 0,C 180,E1 -3702.453,E2 -3702.453} C_VEL
LIN {X 0,Y 546.105,Z 311.576,A -85,B 0,C 180,E1 -3702.874,E2 -3702.874} C_VEL
LIN {X 0,Y 546.245,Z 297.858,A -85,B 0,C 180,E1 -3703.154,E2 -3703.154} C_VEL
LIN {X 0,Y 546.428,Z 201.739,A -85,B 0,C 180,E1 -3704.428,E2 -3704.428} C_VEL
LIN {X 0,Y 545.316,Z 194.247,A -85,B 0,C 180,E1 -3704.579,E2 -3704.579} C_VEL
LIN {X 0,Y 545.546,Z 174.287,A -85,B 0,C 180,E1 -3707.578,E2 -3707.578} C_VEL
LIN {X 0,Y 545.925,Z 154.833,A -85,B 0,C 180,E1 -3710.537,E2 -3710.537} C_VEL
LIN {X 0,Y 546.065,Z 141.908,A -85,B 0,C 180,E1 -3712.528,E2 -3712.528} C_VEL
LIN {X 0,Y 545.047,Z 135.595,A -85,B 0,C 180,E1 -3713.561,E2 -3713.561} C_VEL
LIN {X 0,Y 545.029,Z 135.592,A -85,B 0,C 180,E1 -3716.003,E2 -3716.003} C_VEL
LIN {X 0,Y 545.017,Z 135.594,A -85,B 0,C 180,E1 -3718.734,E2 -3718.734} C_VEL
LIN {X 0,Y 545.044,Z 135.593,A -85,B 0,C 180,E1 -3721.676,E2 -3721.676} C_VEL
LIN {X 0,Y 545.034,Z 135.591,A -85,B 0,C 180,E1 -3724.567,E2 -3724.567} C_VEL
LIN {X 0,Y 544.994,Z 135.601,A -85,B 0,C 180,E1 -3727.308,E2 -3727.308} C_VEL
LIN {X 0,Y 545.005,Z 135.592,A -85,B 0,C 180,E1 -3730.148,E2 -3730.148} C_VEL
LIN {X 0,Y 545.011,Z 135.595,A -85,B 0,C 180,E1 -3732.691,E2 -3732.691} C_VEL
LIN {X 0,Y 545.017,Z 135.598,A -85,B 0,C 180,E1 -3735.172,E2 -3735.172} C_VEL
LIN {X 0,Y 545.023,Z 135.592,A -85,B 0,C 180,E1 -3738.41,E2 -3738.41} C_VEL
LIN {X 0,Y 545.036,Z 135.595,A -85,B 0,C 180,E1 -3740.814,E2 -3740.814} C_VEL
LIN {X 0,Y 545.003,Z 135.592,A -85,B 0,C 180,E1 -3743.616,E2 -3743.616} C_VEL
LIN {X 0,Y 545.025,Z 135.592,A -85,B 0,C 180,E1 -3746.325,E2 -3746.325} C_VEL
LIN {X 0,Y 545.034,Z 135.594,A -85,B 0,C 180,E1 -3748.95,E2 -3748.95} C_VEL
LIN {X 0,Y 545.034,Z 135.587,A -85,B 0,C 180,E1 -3751.504,E2 -3751.504} C_VEL
LIN {X 0,Y 545.031,Z 135.589,A -85,B 0,C 180,E1 -3753.997,E2 -3753.997} C_VEL
LIN {X 0,Y 545.049,Z 135.591,A -85,B 0,C 180,E1 -3756.439,E2 -3756.439} C_VEL
LIN {X 0,Y 545.019,Z 135.592,A -85,B 0,C 180,E1 -3758.835,E2 -3758.835} C_VEL
LIN {X 0,Y 545.004,Z 135.593,A -85,B 0,C 180,E1 -3761.193,E2 -3761.193} C_VEL
LIN {X 0,Y 545.024,Z 135.588,A -85,B 0,C 180,E1 -3763.52,E2 -3763.52} C_VEL
LIN {X 0,Y 545.052,Z 135.587,A -85,B 0,C 180,E1 -3765.819,E2 -3765.819} C_VEL
LIN {X 0,Y 545.075,Z 135.583,A -85,B 0,C 180,E1 -3768.848,E2 -3768.848} C_VEL
LIN {X 0,Y 545.069,Z 135.586,A -85,B 0,C 180,E1 -3771.846,E2 -3771.846} C_VEL
LIN {X 0,Y 545.163,Z 135.573,A -85,B 0,C 180,E1 -3774.823,E2 -3774.823} C_VEL
LIN {X 0,Y 545.192,Z 135.57,A -85,B 0,C 180,E1 -3777.784,E2 -3777.784} C_VEL
LIN {X 0,Y 545.194,Z 135.575,A -85,B 0,C 180,E1 -3780,E2 -3780} C_VEL
LIN {X 0,Y 545.145,Z 135.574,A -85,B 0,C 180,E1 -3782.956,E2 -3782.956} C_VEL
LIN {X 0,Y 545.127,Z 135.584,A -85,B 0,C 180,E1 -3785.92,E2 -3785.92} C_VEL
LIN {X 0,Y 545.071,Z 135.583,A -85,B 0,C 180,E1 -3788.901,E2 -3788.901} C_VEL
LIN {X 0,Y 545.069,Z 135.592,A -85,B 0,C 180,E1 -3791.906,E2 -3791.906} C_VEL
LIN {X 0,Y 545.08,Z 135.583,A -85,B 0,C 180,E1 -3794.944,E2 -3794.944} C_VEL
LIN {X 0,Y 545.045,Z 135.593,A -85,B 0,C 180,E1 -3798.027,E2 -3798.027} C_VEL
LIN {X 0,Y 545.033,Z 135.59,A -85,B 0,C 180,E1 -3800.375,E2 -3800.375} C_VEL
LIN {X 0,Y 544.995,Z 135.593,A -85,B 0,C 180,E1 -3802.76,E2 -3802.76} C_VEL
LIN {X 0,Y 545.04,Z 135.596,A -85,B 0,C 180,E1 -3805.495,E2 -3805.495} C_VEL
LIN {X 0,Y 545.036,Z 135.589,A -85,B 0,C 180,E1 -3808.496,E2 -3808.496} C_VEL
LIN {X 0,Y 545.048,Z 135.595,A -85,B 0,C 180,E1 -3811.676,E2 -3811.676} C_VEL
LIN {X 0,Y 545.049,Z 135.588,A -85,B 0,C 180,E1 -3814.566,E2 -3814.566} C_VEL
LIN {X 0,Y 545.066,Z 135.59,A -85,B 0,C 180,E1 -3816.965,E2 -3816.965} C_VEL
LIN {X 0,Y 544.735,Z 135.935,A -85,B 0,C 180,E1 -3817.373,E2 -3817.373} C_VEL
LIN {X 0,Y 543.449,Z 137.462,A -85,B 0,C 180,E1 -3817.958,E2 -3817.958} C_VEL
LIN {X 0,Y 541.715,Z 139.822,A -85,B 0,C 180,E1 -3818.507,E2 -3818.507} C_VEL
LIN {X 0,Y 539.072,Z 144.894,A -85,B 0,C 180,E1 -3819.403,E2 -3819.403} C_VEL
LIN {X 0,Y 538.506,Z 148.048,A -85,B 0,C 180,E1 -3819.951,E2 -3819.951} C_VEL
LIN {X 0,Y 538.31,Z 163.734,A -85,B 0,C 180,E1 -3822.758,E2 -3822.758} C_VEL
LIN {X 0,Y 538.255,Z 166.697,A -85,B 0,C 180,E1 -3823.291,E2 -3823.291} C_VEL
LIN {X 0,Y 539.686,Z 175.04,A -85,B 0,C 180,E1 -3823.461,E2 -3823.461} C_VEL
LIN {X 0,Y 539.315,Z 273.784,A -85,B 0,C 180,E1 -3824.803,E2 -3824.803} C_VEL
LIN {X 0,Y 539.161,Z 287.263,A -85,B 0,C 180,E1 -3825.144,E2 -3825.144} C_VEL
LIN {X 0,Y 538.989,Z 298.948,A -85,B 0,C 180,E1 -3825.58,E2 -3825.58} C_VEL
LIN {X 0,Y 538.762,Z 310.442,A -85,B 0,C 180,E1 -3826.151,E2 -3826.151} C_VEL
LIN {X 0,Y 538.542,Z 321.156,A -85,B 0,C 180,E1 -3826.835,E2 -3826.835} C_VEL
LIN {X 0,Y 538.318,Z 332.091,A -85,B 0,C 180,E1 -3827.712,E2 -3827.712} C_VEL
LIN {X 0,Y 538.12,Z 341.189,A -85,B 0,C 180,E1 -3828.61,E2 -3828.61} C_VEL
LIN {X 0,Y 537.928,Z 350.208,A -85,B 0,C 180,E1 -3829.705,E2 -3829.705} C_VEL
LIN {X 0,Y 537.784,Z 357.429,A -85,B 0,C 180,E1 -3830.793,E2 -3830.793} C_VEL
LIN {X 0,Y 537.645,Z 364.296,A -85,B 0,C 180,E1 -3832.093,E2 -3832.093} C_VEL
LIN {X 0,Y 537.633,Z 368.215,A -85,B 0,C 180,E1 -3833.035,E2 -3833.035} C_VEL
LIN {X 0,Y 537.548,Z 371.897,A -85,B 0,C 180,E1 -3834.155,E2 -3834.155} C_VEL
LIN {X 0,Y 537.483,Z 374.948,A -85,B 0,C 180,E1 -3835.465,E2 -3835.465} C_VEL
LIN {X 0,Y 537.467,Z 376.778,A -85,B 0,C 180,E1 -3836.812,E2 -3836.812} C_VEL
LIN {X 0,Y 537.455,Z 377.283,A -85,B 0,C 180,E1 -3838.209,E2 -3838.209} C_VEL
LIN {X 0,Y 537.506,Z 376.379,A -85,B 0,C 180,E1 -3839.651,E2 -3839.651} C_VEL
LIN {X 0,Y 537.512,Z 373.842,A -85,B 0,C 180,E1 -3841.167,E2 -3841.167} C_VEL
LIN {X 0,Y 537.573,Z 370.662,A -85,B 0,C 180,E1 -3842.347,E2 -3842.347} C_VEL
LIN {X 0,Y 537.665,Z 365.969,A -85,B 0,C 180,E1 -3843.613,E2 -3843.613} C_VEL
LIN {X 0,Y 537.733,Z 359.904,A -85,B 0,C 180,E1 -3844.864,E2 -3844.864} C_VEL
LIN {X 0,Y 537.878,Z 353.594,A -85,B 0,C 180,E1 -3845.901,E2 -3845.901} C_VEL
LIN {X 0,Y 538.024,Z 345.972,A -85,B 0,C 180,E1 -3846.928,E2 -3846.928} C_VEL
LIN {X 0,Y 538.204,Z 336.184,A -85,B 0,C 180,E1 -3847.993,E2 -3847.993} C_VEL
LIN {X 0,Y 538.436,Z 326.302,A -85,B 0,C 180,E1 -3848.864,E2 -3848.864} C_VEL
LIN {X 0,Y 538.682,Z 315.772,A -85,B 0,C 180,E1 -3849.616,E2 -3849.616} C_VEL
LIN {X 0,Y 538.927,Z 303.903,A -85,B 0,C 180,E1 -3850.28,E2 -3850.28} C_VEL
LIN {X 0,Y 539.085,Z 292.127,A -85,B 0,C 180,E1 -3850.781,E2 -3850.781} C_VEL
LIN {X 0,Y 539.246,Z 278.796,A -85,B 0,C 180,E1 -3851.182,E2 -3851.182} C_VEL
LIN {X 0,Y 539.351,Z 264.362,A -85,B 0,C 180,E1 -3851.432,E2 -3851.432} C_VEL
LIN {X 0,Y 539.56,Z 174.363,A -85,B 0,C 180,E1 -3852.64,E2 -3852.64} C_VEL
LIN {X 0,Y 538.247,Z 166.713,A -85,B 0,C 180,E1 -3852.793,E2 -3852.793} C_VEL
LIN {X 0,Y 538.47,Z 151.167,A -85,B 0,C 180,E1 -3855.642,E2 -3855.642} C_VEL
LIN {X 0,Y 538.635,Z 140.708,A -85,B 0,C 180,E1 -3857.567,E2 -3857.567} C_VEL
LIN {X 0,Y 538.121,Z 136.458,A -85,B 0,C 180,E1 -3858.385,E2 -3858.385} C_VEL
LIN {X 0,Y 538.06,Z 136.459,A -85,B 0,C 180,E1 -3861.739,E2 -3861.739} C_VEL
LIN {X 0,Y 538.149,Z 136.451,A -85,B 0,C 180,E1 -3864.755,E2 -3864.755} C_VEL
LIN {X 0,Y 538.167,Z 136.444,A -85,B 0,C 180,E1 -3867.755,E2 -3867.755} C_VEL
LIN {X 0,Y 538.178,Z 136.446,A -85,B 0,C 180,E1 -3870.748,E2 -3870.748} C_VEL
LIN {X 0,Y 538.121,Z 136.45,A -85,B 0,C 180,E1 -3872.995,E2 -3872.995} C_VEL
LIN {X 0,Y 538.09,Z 136.458,A -85,B 0,C 180,E1 -3875.998,E2 -3875.998} C_VEL
LIN {X 0,Y 538.051,Z 136.458,A -85,B 0,C 180,E1 -3879.018,E2 -3879.018} C_VEL
LIN {X 0,Y 538.062,Z 136.466,A -85,B 0,C 180,E1 -3882.063,E2 -3882.063} C_VEL
LIN {X 0,Y 538.041,Z 136.459,A -85,B 0,C 180,E1 -3885.144,E2 -3885.144} C_VEL
LIN {X 0,Y 538.006,Z 136.468,A -85,B 0,C 180,E1 -3888.271,E2 -3888.271} C_VEL
LIN {X 0,Y 538.031,Z 136.461,A -85,B 0,C 180,E1 -3890.652,E2 -3890.652} C_VEL
LIN {X 0,Y 538.009,Z 136.464,A -85,B 0,C 180,E1 -3893.072,E2 -3893.072} C_VEL
LIN {X 0,Y 537.998,Z 136.472,A -85,B 0,C 180,E1 -3895.662,E2 -3895.662} C_VEL
LIN {X 0,Y 537.995,Z 136.469,A -85,B 0,C 180,E1 -3898.053,E2 -3898.053} C_VEL
LIN {X 0,Y 538.01,Z 136.463,A -85,B 0,C 180,E1 -3900.628,E2 -3900.628} C_VEL
LIN {X 0,Y 538.023,Z 136.466,A -85,B 0,C 180,E1 -3903.279,E2 -3903.279} C_VEL
LIN {X 0,Y 537.991,Z 136.468,A -85,B 0,C 180,E1 -3906.005,E2 -3906.005} C_VEL
LIN {X 0,Y 538.011,Z 136.464,A -85,B 0,C 180,E1 -3908.831,E2 -3908.831} C_VEL
LIN {X 0,Y 537.991,Z 136.468,A -85,B 0,C 180,E1 -3911.874,E2 -3911.874} C_VEL
LIN {X 0,Y 537.997,Z 136.468,A -85,B 0,C 180,E1 -3914.864,E2 -3914.864} C_VEL
LIN {X 0,Y 537.977,Z 136.476,A -85,B 0,C 180,E1 -3917.21,E2 -3917.21} C_VEL
LIN {X 0,Y 538.011,Z 136.463,A -85,B 0,C 180,E1 -3920.202,E2 -3920.202} C_VEL
LIN {X 0,Y 538.022,Z 136.471,A -85,B 0,C 180,E1 -3923.067,E2 -3923.067} C_VEL
LIN {X 0,Y 538.001,Z 136.464,A -85,B 0,C 180,E1 -3925.825,E2 -3925.825} C_VEL
LIN {X 0,Y 537.994,Z 136.468,A -85,B 0,C 180,E1 -3928.497,E2 -3928.497} C_VEL
LIN {X 0,Y 537.988,Z 136.472,A -85,B 0,C 180,E1 -3931.095,E2 -3931.095} C_VEL
LIN {X 0,Y 537.993,Z 136.465,A -85,B 0,C 180,E1 -3933.631,E2 -3933.631} C_VEL
LIN {X 0,Y 537.988,Z 136.467,A -85,B 0,C 180,E1 -3936.128,E2 -3936.128} C_VEL
LIN {X 0,Y 538.003,Z 136.471,A -85,B 0,C 180,E1 -3938.545,E2 -3938.545} C_VEL
LIN {X 0,Y 538.01,Z 136.468,A -85,B 0,C 180,E1 -3940.939,E2 -3940.939} C_VEL
LIN {X 0,Y 537.967,Z 136.469,A -85,B 0,C 180,E1 -3943.297,E2 -3943.297} C_VEL
LIN {X 0,Y 538.039,Z 136.459,A -85,B 0,C 180,E1 -3945.63,E2 -3945.63} C_VEL
LIN {X 0,Y 538.081,Z 136.46,A -85,B 0,C 180,E1 -3948.702,E2 -3948.702} C_VEL
LIN {X 0,Y 538.039,Z 136.46,A -85,B 0,C 180,E1 -3951.739,E2 -3951.739} C_VEL
LIN {X 0,Y 538.125,Z 136.452,A -85,B 0,C 180,E1 -3954.755,E2 -3954.755} C_VEL
LIN {X 0,Y 538.164,Z 136.446,A -85,B 0,C 180,E1 -3957.755,E2 -3957.755} C_VEL
LIN {X 0,Y 538.163,Z 136.45,A -85,B 0,C 180,E1 -3960,E2 -3960} C_VEL
LIN {X 0,Y 538.114,Z 136.45,A -85,B 0,C 180,E1 -3962.995,E2 -3962.995} C_VEL
LIN {X 0,Y 538.083,Z 136.463,A -85,B 0,C 180,E1 -3965.998,E2 -3965.998} C_VEL
LIN {X 0,Y 538.029,Z 136.461,A -85,B 0,C 180,E1 -3969.018,E2 -3969.018} C_VEL
LIN {X 0,Y 538.037,Z 136.466,A -85,B 0,C 180,E1 -3972.064,E2 -3972.064} C_VEL
LIN {X 0,Y 537.991,Z 136.466,A -85,B 0,C 180,E1 -3975.145,E2 -3975.145} C_VEL
LIN {X 0,Y 537.986,Z 136.468,A -85,B 0,C 180,E1 -3978.272,E2 -3978.272} C_VEL
LIN {X 0,Y 537.975,Z 136.467,A -85,B 0,C 180,E1 -3980.654,E2 -3980.654} C_VEL
LIN {X 0,Y 537.978,Z 136.469,A -85,B 0,C 180,E1 -3983.074,E2 -3983.074} C_VEL
LIN {X 0,Y 537.988,Z 136.474,A -85,B 0,C 180,E1 -3985.659,E2 -3985.659} C_VEL
LIN {X 0,Y 537.974,Z 136.469,A -85,B 0,C 180,E1 -3988.054,E2 -3988.054} C_VEL
LIN {X 0,Y 537.99,Z 136.466,A -85,B 0,C 180,E1 -3990.629,E2 -3990.629} C_VEL
LIN {X 0,Y 538.002,Z 136.472,A -85,B 0,C 180,E1 -3993.275,E2 -3993.275} C_VEL
LIN {X 0,Y 537.956,Z 136.47,A -85,B 0,C 180,E1 -3996.008,E2 -3996.008} C_VEL
LIN {X 0,Y 537.987,Z 136.469,A -85,B 0,C 180,E1 -3998.833,E2 -3998.833} C_VEL
LIN {X 0,Y 537.979,Z 136.468,A -85,B 0,C 180,E1 -4001.872,E2 -4001.872} C_VEL
LIN {X 0,Y 537.994,Z 136.471,A -85,B 0,C 180,E1 -4004.864,E2 -4004.864} C_VEL
LIN {X 0,Y 537.972,Z 136.474,A -85,B 0,C 180,E1 -4007.209,E2 -4007.209} C_VEL
LIN {X 0,Y 537.983,Z 136.467,A -85,B 0,C 180,E1 -4010.199,E2 -4010.199} C_VEL
LIN {X 0,Y 537.956,Z 136.476,A -85,B 0,C 180,E1 -4013.061,E2 -4013.061} C_VEL
LIN {X 0,Y 537.989,Z 136.466,A -85,B 0,C 180,E1 -4015.824,E2 -4015.824} C_VEL
LIN {X 0,Y 537.99,Z 136.471,A -85,B 0,C 180,E1 -4018.497,E2 -4018.497} C_VEL
LIN {X 0,Y 537.986,Z 136.471,A -85,B 0,C 180,E1 -4021.095,E2 -4021.095} C_VEL
LIN {X 0,Y 537.977,Z 136.47,A -85,B 0,C 180,E1 -4023.63,E2 -4023.63} C_VEL
LIN {X 0,Y 538.003,Z 136.5,A -85,B 0,C 180,E1 -4026.213,E2 -4026.213} C_VEL
LIN {X 0,Y 539.18,Z 143.768,A -85,B 0,C 180,E1 -4027.426,E2 -4027.426} C_VEL
LIN {X 0,Y 538.855,Z 161.298,A -85,B 0,C 180,E1 -4030.178,E2 -4030.178} C_VEL
LIN {X 0,Y 538.521,Z 179.11,A -85,B 0,C 180,E1 -4032.924,E2 -4032.924} C_VEL
LIN {X 0,Y 538.291,Z 194.234,A -85,B 0,C 180,E1 -4035.238,E2 -4035.238} C_VEL
LIN {X 0,Y 539.63,Z 203.666,A -85,B 0,C 180,E1 -4035.415,E2 -4035.415} C_VEL
LIN {X 0,Y 539.291,Z 303.19,A -85,B 0,C 180,E1 -4036.769,E2 -4036.769} C_VEL
LIN {X 0,Y 539.112,Z 316.206,A -85,B 0,C 180,E1 -4037.1,E2 -4037.1} C_VEL
LIN {X 0,Y 538.923,Z 328.804,A -85,B 0,C 180,E1 -4037.574,E2 -4037.574} C_VEL
LIN {X 0,Y 538.688,Z 339.597,A -85,B 0,C 180,E1 -4038.118,E2 -4038.118} C_VEL
LIN {X 0,Y 538.466,Z 351.638,A -85,B 0,C 180,E1 -4038.9,E2 -4038.9} C_VEL
LIN {X 0,Y 538.232,Z 362.104,A -85,B 0,C 180,E1 -4039.752,E2 -4039.752} C_VEL
LIN {X 0,Y 538.047,Z 370.66,A -85,B 0,C 180,E1 -4040.603,E2 -4040.603} C_VEL
LIN {X 0,Y 537.899,Z 378.553,A -85,B 0,C 180,E1 -4041.547,E2 -4041.547} C_VEL
LIN {X 0,Y 537.755,Z 386.26,A -85,B 0,C 180,E1 -4042.679,E2 -4042.679} C_VEL
LIN {X 0,Y 537.685,Z 393.362,A -85,B 0,C 180,E1 -4043.998,E2 -4043.998} C_VEL
LIN {X 0,Y 537.54,Z 398.084,A -85,B 0,C 180,E1 -4045.125,E2 -4045.125} C_VEL
LIN {X 0,Y 537.591,Z 401.694,A -85,B 0,C 180,E1 -4046.252,E2 -4046.252} C_VEL
LIN {X 0,Y 537.551,Z 403.554,A -85,B 0,C 180,E1 -4047.002,E2 -4047.002} C_VEL
LIN {X 0,Y 537.451,Z 405.943,A -85,B 0,C 180,E1 -4048.501,E2 -4048.501} C_VEL
LIN {X 0,Y 537.445,Z 406.766,A -85,B 0,C 180,E1 -4050,E2 -4050} C_VEL
LIN {X 0,Y 537.451,Z 405.942,A -85,B 0,C 180,E1 -4051.499,E2 -4051.499} C_VEL
LIN {X 0,Y 537.49,Z 404.948,A -85,B 0,C 180,E1 -4052.248,E2 -4052.248} C_VEL
LIN {X 0,Y 537.551,Z 403.553,A -85,B 0,C 180,E1 -4052.998,E2 -4052.998} C_VEL
LIN {X 0,Y 537.603,Z 400.618,A -85,B 0,C 180,E1 -4054.123,E2 -4054.123} C_VEL
LIN {X 0,Y 537.587,Z 396.641,A -85,B 0,C 180,E1 -4055.251,E2 -4055.251} C_VEL
LIN {X 0,Y 537.619,Z 391.862,A -85,B 0,C 180,E1 -4056.311,E2 -4056.311} C_VEL
LIN {X 0,Y 537.755,Z 385.08,A -85,B 0,C 180,E1 -4057.51,E2 -4057.51} C_VEL
LIN {X 0,Y 537.914,Z 377.04,A -85,B 0,C 180,E1 -4058.642,E2 -4058.642} C_VEL
LIN {X 0,Y 538.071,Z 368.845,A -85,B 0,C 180,E1 -4059.586,E2 -4059.586} C_VEL
LIN {X 0,Y 538.336,Z 358.85,A -85,B 0,C 180,E1 -4060.531,E2 -4060.531} C_VEL
LIN {X 0,Y 538.541,Z 348.982,A -85,B 0,C 180,E1 -4061.289,E2 -4061.289} C_VEL
LIN {X 0,Y 538.719,Z 337.902,A -85,B 0,C 180,E1 -4061.972,E2 -4061.972} C_VEL
LIN {X 0,Y 538.952,Z 325.344,A -85,B 0,C 180,E1 -4062.569,E2 -4062.569} C_VEL
LIN {X 0,Y 539.169,Z 313.063,A -85,B 0,C 180,E1 -4062.994,E2 -4062.994} C_VEL
LIN {X 0,Y 539.318,Z 300.505,A -85,B 0,C 180,E1 -4063.278,E2 -4063.278} C_VEL
LIN {X 0,Y 539.546,Z 202.58,A -85,B 0,C 180,E1 -4064.601,E2 -4064.601} C_VEL
LIN {X 0,Y 538.25,Z 194.092,A -85,B 0,C 180,E1 -4064.766,E2 -4064.766} C_VEL
LIN {X 0,Y 538.524,Z 176.329,A -85,B 0,C 180,E1 -4067.467,E2 -4067.467} C_VEL
LIN {X 0,Y 538.828,Z 160.996,A -85,B 0,C 180,E1 -4069.824,E2 -4069.824} C_VEL
LIN {X 0,Y 539.112,Z 143.05,A -85,B 0,C 180,E1 -4072.617,E2 -4072.617} C_VEL
LIN {X 0,Y 537.998,Z 136.473,A -85,B 0,C 180,E1 -4073.731,E2 -4073.731} C_VEL
LIN {X 0,Y 537.977,Z 136.469,A -85,B 0,C 180,E1 -4076.37,E2 -4076.37} C_VEL
LIN {X 0,Y 537.975,Z 136.473,A -85,B 0,C 180,E1 -4078.922,E2 -4078.922} C_VEL
LIN {X 0,Y 537.995,Z 136.469,A -85,B 0,C 180,E1 -4081.884,E2 -4081.884} C_VEL
LIN {X 0,Y 537.984,Z 136.469,A -85,B 0,C 180,E1 -4084.613,E2 -4084.613} C_VEL
LIN {X 0,Y 537.96,Z 136.471,A -85,B 0,C 180,E1 -4087.881,E2 -4087.881} C_VEL
LIN {X 0,Y 537.953,Z 136.476,A -85,B 0,C 180,E1 -4090.785,E2 -4090.785} C_VEL
LIN {X 0,Y 537.98,Z 136.468,A -85,B 0,C 180,E1 -4093.819,E2 -4093.819} C_VEL
LIN {X 0,Y 537.98,Z 136.468,A -85,B 0,C 180,E1 -4096.181,E2 -4096.181} C_VEL
LIN {X 0,Y 537.954,Z 136.474,A -85,B 0,C 180,E1 -4099.265,E2 -4099.265} C_VEL
LIN {X 0,Y 537.966,Z 136.469,A -85,B 0,C 180,E1 -4102.12,E2 -4102.12} C_VEL
LIN {X 0,Y 537.986,Z 136.468,A -85,B 0,C 180,E1 -4105.387,E2 -4105.387} C_VEL
LIN {X 0,Y 537.996,Z 136.465,A -85,B 0,C 180,E1 -4108.116,E2 -4108.116} C_VEL
LIN {X 0,Y 537.988,Z 136.468,A -85,B 0,C 180,E1 -4111.096,E2 -4111.096} C_VEL
LIN {X 0,Y 537.979,Z 136.467,A -85,B 0,C 180,E1 -4113.63,E2 -4113.63} C_VEL
LIN {X 0,Y 537.987,Z 136.467,A -85,B 0,C 180,E1 -4116.128,E2 -4116.128} C_VEL
LIN {X 0,Y 537.992,Z 136.473,A -85,B 0,C 180,E1 -4118.545,E2 -4118.545} C_VEL
LIN {X 0,Y 537.96,Z 136.473,A -85,B 0,C 180,E1 -4120.937,E2 -4120.937} C_VEL
LIN {X 0,Y 537.972,Z 136.467,A -85,B 0,C 180,E1 -4123.297,E2 -4123.297} C_VEL
LIN {X 0,Y 538.025,Z 136.461,A -85,B 0,C 180,E1 -4125.63,E2 -4125.63} C_VEL
LIN {X 0,Y 538.027,Z 136.463,A -85,B 0,C 180,E1 -4128.7,E2 -4128.7} C_VEL
LIN {X 0,Y 538.038,Z 136.461,A -85,B 0,C 180,E1 -4131.739,E2 -4131.739} C_VEL
LIN {X 0,Y 538.122,Z 136.451,A -85,B 0,C 180,E1 -4134.755,E2 -4134.755} C_VEL
LIN {X 0,Y 538.164,Z 136.445,A -85,B 0,C 180,E1 -4137.755,E2 -4137.755} C_VEL
LIN {X 0,Y 538.163,Z 136.45,A -85,B 0,C 180,E1 -4140,E2 -4140} C_VEL
LIN {X 0,Y 538.113,Z 136.45,A -85,B 0,C 180,E1 -4142.995,E2 -4142.995} C_VEL
LIN {X 0,Y 538.083,Z 136.461,A -85,B 0,C 180,E1 -4145.998,E2 -4145.998} C_VEL
LIN {X 0,Y 538.029,Z 136.46,A -85,B 0,C 180,E1 -4149.018,E2 -4149.018} C_VEL
LIN {X 0,Y 538.04,Z 136.466,A -85,B 0,C 180,E1 -4152.064,E2 -4152.064} C_VEL
LIN {X 0,Y 538.041,Z 136.46,A -85,B 0,C 180,E1 -4155.144,E2 -4155.144} C_VEL
LIN {X 0,Y 537.998,Z 136.467,A -85,B 0,C 180,E1 -4158.271,E2 -4158.271} C_VEL
LIN {X 0,Y 537.991,Z 136.466,A -85,B 0,C 180,E1 -4160.653,E2 -4160.653} C_VEL
LIN {X 0,Y 537.984,Z 136.468,A -85,B 0,C 180,E1 -4163.073,E2 -4163.073} C_VEL
LIN {X 0,Y 537.998,Z 136.474,A -85,B 0,C 180,E1 -4165.661,E2 -4165.661} C_VEL
LIN {X 0,Y 537.989,Z 136.47,A -85,B 0,C 180,E1 -4168.053,E2 -4168.053} C_VEL
LIN {X 0,Y 537.996,Z 136.466,A -85,B 0,C 180,E1 -4170.629,E2 -4170.629} C_VEL
LIN {X 0,Y 538.024,Z 136.469,A -85,B 0,C 180,E1 -4173.278,E2 -4173.278} C_VEL
LIN {X 0,Y 537.991,Z 136.471,A -85,B 0,C 180,E1 -4176.005,E2 -4176.005} C_VEL
LIN {X 0,Y 538.072,Z 136.622,A -85,B 0,C 180,E1 -4177.871,E2 -4177.871} C_VEL
LIN {X 0,Y 538.537,Z 141.588,A -85,B 0,C 180,E1 -4178.786,E2 -4178.786} C_VEL
LIN {X 0,Y 538.506,Z 148.048,A -85,B 0,C 180,E1 -4179.951,E2 -4179.951} C_VEL
LIN {X 0,Y 537.874,Z 151.146,A -85,B 0,C 180,E1 -4180.482,E2 -4180.482} C_VEL
LIN {X 0,Y 534.973,Z 156.424,A -85,B 0,C 180,E1 -4181.325,E2 -4181.325} C_VEL
LIN {X 0,Y 532.013,Z 161.68,A -85,B 0,C 180,E1 -4182.176,E2 -4182.176} C_VEL
LIN {X 0,Y 531.31,Z 164.79,A -85,B 0,C 180,E1 -4182.715,E2 -4182.715} C_VEL
LIN {X 0,Y 531.276,Z 167.061,A -85,B 0,C 180,E1 -4183.111,E2 -4183.111} C_VEL
LIN {X 0,Y 532.836,Z 175.759,A -85,B 0,C 180,E1 -4183.277,E2 -4183.277} C_VEL
LIN {X 0,Y 532.397,Z 274.18,A -85,B 0,C 180,E1 -4184.634,E2 -4184.634} C_VEL
LIN {X 0,Y 532.245,Z 287.302,A -85,B 0,C 180,E1 -4184.971,E2 -4184.971} C_VEL
LIN {X 0,Y 532.06,Z 299.841,A -85,B 0,C 180,E1 -4185.447,E2 -4185.447} C_VEL
LIN {X 0,Y 531.793,Z 311.82,A -85,B 0,C 180,E1 -4186.066,E2 -4186.066} C_VEL
LIN {X 0,Y 531.521,Z 323.686,A -85,B 0,C 180,E1 -4186.863,E2 -4186.863} C_VEL
LIN {X 0,Y 531.294,Z 333.904,A -85,B 0,C 180,E1 -4187.722,E2 -4187.722} C_VEL
LIN {X 0,Y 531.088,Z 342.187,A -85,B 0,C 180,E1 -4188.573,E2 -4188.573} C_VEL
LIN {X 0,Y 530.9,Z 350.147,A -85,B 0,C 180,E1 -4189.559,E2 -4189.559} C_VEL
LIN {X 0,Y 530.717,Z 358.006,A -85,B 0,C 180,E1 -4190.763,E2 -4190.763} C_VEL
LIN {X 0,Y 530.578,Z 364.326,A -85,B 0,C 180,E1 -4191.98,E2 -4191.98} C_VEL
LIN {X 0,Y 530.56,Z 368.608,A -85,B 0,C 180,E1 -4193.022,E2 -4193.022} C_VEL
LIN {X 0,Y 530.438,Z 372.751,A -85,B 0,C 180,E1 -4194.34,E2 -4194.34} C_VEL
LIN {X 0,Y 530.39,Z 374.83,A -85,B 0,C 180,E1 -4195.265,E2 -4195.265} C_VEL
LIN {X 0,Y 530.364,Z 376.77,A -85,B 0,C 180,E1 -4196.599,E2 -4196.599} C_VEL
LIN {X 0,Y 530.379,Z 377.502,A -85,B 0,C 180,E1 -4198.001,E2 -4198.001} C_VEL
LIN {X 0,Y 530.384,Z 376.793,A -85,B 0,C 180,E1 -4199.463,E2 -4199.463} C_VEL
LIN {X 0,Y 530.415,Z 374.51,A -85,B 0,C 180,E1 -4200.986,E2 -4200.986} C_VEL
LIN {X 0,Y 530.5,Z 370.946,A -85,B 0,C 180,E1 -4202.375,E2 -4202.375} C_VEL
LIN {X 0,Y 530.607,Z 366.275,A -85,B 0,C 180,E1 -4203.659,E2 -4203.659} C_VEL
LIN {X 0,Y 530.657,Z 360.247,A -85,B 0,C 180,E1 -4204.925,E2 -4204.925} C_VEL
LIN {X 0,Y 530.819,Z 353.298,A -85,B 0,C 180,E1 -4206.079,E2 -4206.079} C_VEL
LIN {X 0,Y 531.001,Z 344.663,A -85,B 0,C 180,E1 -4207.223,E2 -4207.223} C_VEL
LIN {X 0,Y 531.258,Z 334.993,A -85,B 0,C 180,E1 -4208.259,E2 -4208.259} C_VEL
LIN {X 0,Y 531.48,Z 325.558,A -85,B 0,C 180,E1 -4209.082,E2 -4209.082} C_VEL
LIN {X 0,Y 531.728,Z 315.608,A -85,B 0,C 180,E1 -4209.79,E2 -4209.79} C_VEL
LIN {X 0,Y 531.996,Z 303.574,A -85,B 0,C 180,E1 -4210.464,E2 -4210.464} C_VEL
LIN {X 0,Y 532.179,Z 291.622,A -85,B 0,C 180,E1 -4210.972,E2 -4210.972} C_VEL
LIN {X 0,Y 532.342,Z 278.976,A -85,B 0,C 180,E1 -4211.353,E2 -4211.353} C_VEL
LIN {X 0,Y 532.471,Z 263.957,A -85,B 0,C 180,E1 -4211.614,E2 -4211.614} C_VEL
LIN {X 0,Y 532.827,Z 175.923,A -85,B 0,C 180,E1 -4212.81,E2 -4212.81} C_VEL
LIN {X 0,Y 531.24,Z 166.965,A -85,B 0,C 180,E1 -4212.98,E2 -4212.98} C_VEL
LIN {X 0,Y 531.478,Z 152.534,A -85,B 0,C 180,E1 -4215.644,E2 -4215.644} C_VEL
LIN {X 0,Y 531.655,Z 142.052,A -85,B 0,C 180,E1 -4217.595,E2 -4217.595} C_VEL
LIN {X 0,Y 531.064,Z 137.338,A -85,B 0,C 180,E1 -4218.514,E2 -4218.514} C_VEL
LIN {X 0,Y 531.036,Z 137.334,A -85,B 0,C 180,E1 -4221.629,E2 -4221.629} C_VEL
LIN {X 0,Y 531.107,Z 137.329,A -85,B 0,C 180,E1 -4224.685,E2 -4224.685} C_VEL
LIN {X 0,Y 531.139,Z 137.32,A -85,B 0,C 180,E1 -4227.725,E2 -4227.725} C_VEL
LIN {X 0,Y 531.149,Z 137.321,A -85,B 0,C 180,E1 -4230.758,E2 -4230.758} C_VEL
LIN {X 0,Y 531.062,Z 137.329,A -85,B 0,C 180,E1 -4233.034,E2 -4233.034} C_VEL
LIN {X 0,Y 531.047,Z 137.337,A -85,B 0,C 180,E1 -4236.078,E2 -4236.078} C_VEL
LIN {X 0,Y 531.013,Z 137.334,A -85,B 0,C 180,E1 -4239.139,E2 -4239.139} C_VEL
LIN {X 0,Y 531.053,Z 137.333,A -85,B 0,C 180,E1 -4241.671,E2 -4241.671} C_VEL
LIN {X 0,Y 531.026,Z 137.333,A -85,B 0,C 180,E1 -4244.952,E2 -4244.952} C_VEL
LIN {X 0,Y 530.974,Z 137.345,A -85,B 0,C 180,E1 -4247.724,E2 -4247.724} C_VEL
LIN {X 0,Y 531.016,Z 137.34,A -85,B 0,C 180,E1 -4250.128,E2 -4250.128} C_VEL
LIN {X 0,Y 530.944,Z 137.344,A -85,B 0,C 180,E1 -4252.574,E2 -4252.574} C_VEL
LIN {X 0,Y 530.952,Z 137.343,A -85,B 0,C 180,E1 -4255.06,E2 -4255.06} C_VEL
LIN {X 0,Y 530.962,Z 137.348,A -85,B 0,C 180,E1 -4257.599,E2 -4257.599} C_VEL
LIN {X 0,Y 530.964,Z 137.341,A -85,B 0,C 180,E1 -4260.643,E2 -4260.643} C_VEL
LIN {X 0,Y 530.964,Z 137.349,A -85,B 0,C 180,E1 -4263.499,E2 -4263.499} C_VEL
LIN {X 0,Y 530.953,Z 137.342,A -85,B 0,C 180,E1 -4266.559,E2 -4266.559} C_VEL
LIN {X 0,Y 530.985,Z 137.347,A -85,B 0,C 180,E1 -4269.444,E2 -4269.444} C_VEL
LIN {X 0,Y 530.921,Z 137.346,A -85,B 0,C 180,E1 -4272.463,E2 -4272.463} C_VEL
LIN {X 0,Y 530.967,Z 137.347,A -85,B 0,C 180,E1 -4275.451,E2 -4275.451} C_VEL
LIN {X 0,Y 530.961,Z 137.342,A -85,B 0,C 180,E1 -4278.561,E2 -4278.561} C_VEL
LIN {X 0,Y 530.955,Z 137.345,A -85,B 0,C 180,E1 -4281.529,E2 -4281.529} C_VEL
LIN {X 0,Y 530.95,Z 137.343,A -85,B 0,C 180,E1 -4284.379,E2 -4284.379} C_VEL
LIN {X 0,Y 530.968,Z 137.347,A -85,B 0,C 180,E1 -4287.133,E2 -4287.133} C_VEL
LIN {X 0,Y 530.938,Z 137.344,A -85,B 0,C 180,E1 -4289.801,E2 -4289.801} C_VEL
LIN {X 0,Y 530.966,Z 137.344,A -85,B 0,C 180,E1 -4292.478,E2 -4292.478} C_VEL
LIN {X 0,Y 530.951,Z 137.349,A -85,B 0,C 180,E1 -4294.94,E2 -4294.94} C_VEL
LIN {X 0,Y 530.956,Z 137.344,A -85,B 0,C 180,E1 -4298.246,E2 -4298.246} C_VEL
LIN {X 0,Y 530.967,Z 137.349,A -85,B 0,C 180,E1 -4300.676,E2 -4300.676} C_VEL
LIN {X 0,Y 530.932,Z 137.347,A -85,B 0,C 180,E1 -4303.069,E2 -4303.069} C_VEL
LIN {X 0,Y 531.001,Z 137.336,A -85,B 0,C 180,E1 -4305.435,E2 -4305.435} C_VEL
LIN {X 0,Y 531.039,Z 137.339,A -85,B 0,C 180,E1 -4308.55,E2 -4308.55} C_VEL
LIN {X 0,Y 530.987,Z 137.338,A -85,B 0,C 180,E1 -4311.628,E2 -4311.628} C_VEL
LIN {X 0,Y 531.086,Z 137.329,A -85,B 0,C 180,E1 -4314.685,E2 -4314.685} C_VEL
LIN {X 0,Y 531.136,Z 137.321,A -85,B 0,C 180,E1 -4317.725,E2 -4317.725} C_VEL
LIN {X 0,Y 531.132,Z 137.326,A -85,B 0,C 180,E1 -4320,E2 -4320} C_VEL
LIN {X 0,Y 531.137,Z 137.326,A -85,B 0,C 180,E1 -4322.275,E2 -4322.275} C_VEL
LIN {X 0,Y 531.084,Z 137.326,A -85,B 0,C 180,E1 -4325.315,E2 -4325.315} C_VEL
LIN {X 0,Y 530.986,Z 137.341,A -85,B 0,C 180,E1 -4328.372,E2 -4328.372} C_VEL
LIN {X 0,Y 531.016,Z 137.34,A -85,B 0,C 180,E1 -4331.65,E2 -4331.65} C_VEL
LIN {X 0,Y 530.967,Z 137.34,A -85,B 0,C 180,E1 -4334.928,E2 -4334.928} C_VEL
LIN {X 0,Y 530.973,Z 137.348,A -85,B 0,C 180,E1 -4337.724,E2 -4337.724} C_VEL
LIN {X 0,Y 530.933,Z 137.345,A -85,B 0,C 180,E1 -4340.941,E2 -4340.941} C_VEL
LIN {X 0,Y 530.925,Z 137.351,A -85,B 0,C 180,E1 -4343.398,E2 -4343.398} C_VEL
LIN {X 0,Y 530.932,Z 137.349,A -85,B 0,C 180,E1 -4345.902,E2 -4345.902} C_VEL
LIN {X 0,Y 530.933,Z 137.344,A -85,B 0,C 180,E1 -4348.459,E2 -4348.459} C_VEL
LIN {X 0,Y 530.938,Z 137.348,A -85,B 0,C 180,E1 -4351.081,E2 -4351.081} C_VEL
LIN {X 0,Y 530.934,Z 137.348,A -85,B 0,C 180,E1 -4353.777,E2 -4353.777} C_VEL
LIN {X 0,Y 530.907,Z 137.348,A -85,B 0,C 180,E1 -4356.562,E2 -4356.562} C_VEL
LIN {X 0,Y 530.946,Z 137.349,A -85,B 0,C 180,E1 -4359.447,E2 -4359.447} C_VEL
LIN {X 0,Y 530.914,Z 137.348,A -85,B 0,C 180,E1 -4362.463,E2 -4362.463} C_VEL
LIN {X 0,Y 530.965,Z 137.344,A -85,B 0,C 180,E1 -4365.45,E2 -4365.45} C_VEL
LIN {X 0,Y 530.949,Z 137.345,A -85,B 0,C 180,E1 -4368.56,E2 -4368.56} C_VEL
LIN {X 0,Y 530.93,Z 137.346,A -85,B 0,C 180,E1 -4371.527,E2 -4371.527} C_VEL
LIN {X 0,Y 530.926,Z 137.348,A -85,B 0,C 180,E1 -4374.377,E2 -4374.377} C_VEL
LIN {X 0,Y 530.946,Z 137.347,A -85,B 0,C 180,E1 -4377.132,E2 -4377.132} C_VEL
LIN {X 0,Y 530.93,Z 137.346,A -85,B 0,C 180,E1 -4379.8,E2 -4379.8} C_VEL
LIN {X 0,Y 530.955,Z 137.349,A -85,B 0,C 180,E1 -4382.48,E2 -4382.48} C_VEL
LIN {X 0,Y 530.935,Z 137.353,A -85,B 0,C 180,E1 -4384.939,E2 -4384.939} C_VEL
LIN {X 0,Y 530.956,Z 137.44,A -85,B 0,C 180,E1 -4386.058,E2 -4386.058} C_VEL
LIN {X 0,Y 532.204,Z 144.628,A -85,B 0,C 180,E1 -4387.278,E2 -4387.278} C_VEL
LIN {X 0,Y 531.902,Z 161.126,A -85,B 0,C 180,E1 -4389.907,E2 -4389.907} C_VEL
LIN {X 0,Y 531.54,Z 177.654,A -85,B 0,C 180,E1 -4392.494,E2 -4392.494} C_VEL
LIN {X 0,Y 531.27,Z 194.13,A -85,B 0,C 180,E1 -4395.051,E2 -4395.051} C_VEL
LIN {X 0,Y 532.78,Z 204.487,A -85,B 0,C 180,E1 -4395.237,E2 -4395.237} C_VEL
LIN {X 0,Y 532.377,Z 302.892,A -85,B 0,C 180,E1 -4396.594,E2 -4396.594} C_VEL
LIN {X 0,Y 532.182,Z 316.703,A -85,B 0,C 180,E1 -4396.953,E2 -4396.953} C_VEL
LIN {X 0,Y 531.951,Z 329.602,A -85,B 0,C 180,E1 -4397.457,E2 -4397.457} C_VEL
LIN {X 0,Y 531.644,Z 342.146,A -85,B 0,C 180,E1 -4398.127,E2 -4398.127} C_VEL
LIN {X 0,Y 531.439,Z 352.711,A -85,B 0,C 180,E1 -4398.848,E2 -4398.848} C_VEL
LIN {X 0,Y 531.176,Z 362.939,A -85,B 0,C 180,E1 -4399.711,E2 -4399.711} C_VEL
LIN {X 0,Y 530.961,Z 372.134,A -85,B 0,C 180,E1 -4400.668,E2 -4400.668} C_VEL
LIN {X 0,Y 530.775,Z 381.09,A -85,B 0,C 180,E1 -4401.817,E2 -4401.817} C_VEL
LIN {X 0,Y 530.622,Z 388.298,A -85,B 0,C 180,E1 -4402.963,E2 -4402.963} C_VEL
LIN {X 0,Y 530.574,Z 394.861,A -85,B 0,C 180,E1 -4404.298,E2 -4404.298} C_VEL
LIN {X 0,Y 530.45,Z 399.2,A -85,B 0,C 180,E1 -4405.44,E2 -4405.44} C_VEL
LIN {X 0,Y 530.516,Z 401.499,A -85,B 0,C 180,E1 -4406.202,E2 -4406.202} C_VEL
LIN {X 0,Y 530.457,Z 403.36,A -85,B 0,C 180,E1 -4406.962,E2 -4406.962} C_VEL
LIN {X 0,Y 530.411,Z 404.754,A -85,B 0,C 180,E1 -4407.722,E2 -4407.722} C_VEL
LIN {X 0,Y 530.347,Z 406.356,A -85,B 0,C 180,E1 -4409.241,E2 -4409.241} C_VEL
LIN {X 0,Y 530.348,Z 406.572,A -85,B 0,C 180,E1 -4410,E2 -4410} C_VEL
LIN {X 0,Y 530.361,Z 405.747,A -85,B 0,C 180,E1 -4411.519,E2 -4411.519} C_VEL
LIN {X 0,Y 530.411,Z 404.752,A -85,B 0,C 180,E1 -4412.278,E2 -4412.278} C_VEL
LIN {X 0,Y 530.457,Z 403.355,A -85,B 0,C 180,E1 -4413.038,E2 -4413.038} C_VEL
LIN {X 0,Y 530.521,Z 400.417,A -85,B 0,C 180,E1 -4414.178,E2 -4414.178} C_VEL
LIN {X 0,Y 530.522,Z 396.438,A -85,B 0,C 180,E1 -4415.321,E2 -4415.321} C_VEL
LIN {X 0,Y 530.583,Z 390.787,A -85,B 0,C 180,E1 -4416.567,E2 -4416.567} C_VEL
LIN {X 0,Y 530.705,Z 383.629,A -85,B 0,C 180,E1 -4417.801,E2 -4417.801} C_VEL
LIN {X 0,Y 530.888,Z 375.327,A -85,B 0,C 180,E1 -4418.949,E2 -4418.949} C_VEL
LIN {X 0,Y 531.067,Z 366.812,A -85,B 0,C 180,E1 -4419.906,E2 -4419.906} C_VEL
LIN {X 0,Y 531.357,Z 356.293,A -85,B 0,C 180,E1 -4420.864,E2 -4420.864} C_VEL
LIN {X 0,Y 531.611,Z 344.47,A -85,B 0,C 180,E1 -4421.726,E2 -4421.726} C_VEL
LIN {X 0,Y 531.899,Z 332.513,A -85,B 0,C 180,E1 -4422.399,E2 -4422.399} C_VEL
LIN {X 0,Y 532.113,Z 320.092,A -85,B 0,C 180,E1 -4422.927,E2 -4422.927} C_VEL
LIN {X 0,Y 532.324,Z 307.29,A -85,B 0,C 180,E1 -4423.31,E2 -4423.31} C_VEL
LIN {X 0,Y 532.466,Z 293.745,A -85,B 0,C 180,E1 -4423.549,E2 -4423.549} C_VEL
LIN {X 0,Y 532.62,Z 202.97,A -85,B 0,C 180,E1 -4424.787,E2 -4424.787} C_VEL
LIN {X 0,Y 531.243,Z 193.87,A -85,B 0,C 180,E1 -4424.967,E2 -4424.967} C_VEL
LIN {X 0,Y 531.582,Z 175.229,A -85,B 0,C 180,E1 -4427.841,E2 -4427.841} C_VEL
LIN {X 0,Y 531.994,Z 155.651,A -85,B 0,C 180,E1 -4430.897,E2 -4430.897} C_VEL
LIN {X 0,Y 532.154,Z 144.101,A -85,B 0,C 180,E1 -4432.724,E2 -4432.724} C_VEL
LIN {X 0,Y 530.94,Z 137.351,A -85,B 0,C 180,E1 -4433.897,E2 -4433.897} C_VEL
LIN {X 0,Y 530.942,Z 137.347,A -85,B 0,C 180,E1 -4436.747,E2 -4436.747} C_VEL
LIN {X 0,Y 530.916,Z 137.357,A -85,B 0,C 180,E1 -4439.327,E2 -4439.327} C_VEL
LIN {X 0,Y 530.95,Z 137.346,A -85,B 0,C 180,E1 -4442.097,E2 -4442.097} C_VEL
LIN {X 0,Y 530.948,Z 137.348,A -85,B 0,C 180,E1 -4444.847,E2 -4444.847} C_VEL
LIN {X 0,Y 530.9,Z 137.354,A -85,B 0,C 180,E1 -4447.514,E2 -4447.514} C_VEL
LIN {X 0,Y 530.907,Z 137.35,A -85,B 0,C 180,E1 -4450.44,E2 -4450.44} C_VEL
LIN {X 0,Y 530.922,Z 137.35,A -85,B 0,C 180,E1 -4453.5,E2 -4453.5} C_VEL
LIN {X 0,Y 530.964,Z 137.343,A -85,B 0,C 180,E1 -4455.624,E2 -4455.624} C_VEL
LIN {X 0,Y 530.91,Z 137.351,A -85,B 0,C 180,E1 -4458.556,E2 -4458.556} C_VEL
LIN {X 0,Y 530.924,Z 137.348,A -85,B 0,C 180,E1 -4461.526,E2 -4461.526} C_VEL
LIN {X 0,Y 530.926,Z 137.347,A -85,B 0,C 180,E1 -4464.378,E2 -4464.378} C_VEL
LIN {X 0,Y 530.946,Z 137.346,A -85,B 0,C 180,E1 -4467.132,E2 -4467.132} C_VEL
LIN {X 0,Y 530.932,Z 137.344,A -85,B 0,C 180,E1 -4469.801,E2 -4469.801} C_VEL
LIN {X 0,Y 530.957,Z 137.347,A -85,B 0,C 180,E1 -4472.48,E2 -4472.48} C_VEL
LIN {X 0,Y 530.936,Z 137.347,A -85,B 0,C 180,E1 -4474.939,E2 -4474.939} C_VEL
LIN {X 0,Y 530.962,Z 137.342,A -85,B 0,C 180,E1 -4477.904,E2 -4477.904} C_VEL
LIN {X 0,Y 530.919,Z 137.354,A -85,B 0,C 180,E1 -4480.674,E2 -4480.674} C_VEL
LIN {X 0,Y 530.935,Z 137.345,A -85,B 0,C 180,E1 -4483.069,E2 -4483.069} C_VEL
LIN {X 0,Y 530.978,Z 137.338,A -85,B 0,C 180,E1 -4485.435,E2 -4485.435} C_VEL
LIN {X 0,Y 530.99,Z 137.341,A -85,B 0,C 180,E1 -4488.549,E2 -4488.549} C_VEL
LIN {X 0,Y 530.985,Z 137.339,A -85,B 0,C 180,E1 -4491.628,E2 -4491.628} C_VEL
LIN {X 0,Y 531.083,Z 137.328,A -85,B 0,C 180,E1 -4494.685,E2 -4494.685} C_VEL
LIN {X 0,Y 531.135,Z 137.32,A -85,B 0,C 180,E1 -4497.725,E2 -4497.725} C_VEL
LIN {X 0,Y 531.131,Z 137.326,A -85,B 0,C 180,E1 -4500,E2 -4500} C_VEL
LIN {X 0,Y 531.136,Z 137.326,A -85,B 0,C 180,E1 -4502.275,E2 -4502.275} C_VEL
LIN {X 0,Y 531.085,Z 137.326,A -85,B 0,C 180,E1 -4505.315,E2 -4505.315} C_VEL
LIN {X 0,Y 530.987,Z 137.341,A -85,B 0,C 180,E1 -4508.372,E2 -4508.372} C_VEL
LIN {X 0,Y 531.016,Z 137.34,A -85,B 0,C 180,E1 -4511.65,E2 -4511.65} C_VEL
LIN {X 0,Y 531.024,Z 137.334,A -85,B 0,C 180,E1 -4514.95,E2 -4514.95} C_VEL
LIN {X 0,Y 530.975,Z 137.348,A -85,B 0,C 180,E1 -4517.724,E2 -4517.724} C_VEL
LIN {X 0,Y 530.975,Z 137.343,A -85,B 0,C 180,E1 -4520.129,E2 -4520.129} C_VEL
LIN {X 0,Y 530.923,Z 137.347,A -85,B 0,C 180,E1 -4522.575,E2 -4522.575} C_VEL
LIN {X 0,Y 530.953,Z 137.345,A -85,B 0,C 180,E1 -4525.06,E2 -4525.06} C_VEL
LIN {X 0,Y 530.959,Z 137.351,A -85,B 0,C 180,E1 -4527.599,E2 -4527.599} C_VEL
LIN {X 0,Y 530.951,Z 137.344,A -85,B 0,C 180,E1 -4530.64,E2 -4530.64} C_VEL
LIN {X 0,Y 530.965,Z 137.349,A -85,B 0,C 180,E1 -4533.499,E2 -4533.499} C_VEL
LIN {X 0,Y 530.955,Z 137.346,A -85,B 0,C 180,E1 -4536.559,E2 -4536.559} C_VEL
LIN {X 0,Y 531.034,Z 137.423,A -85,B 0,C 180,E1 -4537.742,E2 -4537.742} C_VEL
LIN {X 0,Y 531.567,Z 142.768,A -85,B 0,C 180,E1 -4538.734,E2 -4538.734} C_VEL
LIN {X 0,Y 531.403,Z 157.497,A -85,B 0,C 180,E1 -4541.397,E2 -4541.397} C_VEL
LIN {X 0,Y 531.31,Z 164.79,A -85,B 0,C 180,E1 -4542.715,E2 -4542.715} C_VEL
LIN {X 0,Y 530.909,Z 166.639,A -85,B 0,C 180,E1 -4542.919,E2 -4542.919} C_VEL
LIN {X 0,Y 529.662,Z 169.825,A -85,B 0,C 180,E1 -4543.067,E2 -4543.067} C_VEL
LIN {X 0,Y 527,Z 176.289,A -85,B 0,C 180,E1 -4543.114,E2 -4543.114} C_VEL
LIN {X 0,Y 526.053,Z 180.363,A -85,B 0,C 180,E1 -4543.138,E2 -4543.138} C_VEL
LIN {X 0,Y 525.725,Z 186.815,A -85,B 0,C 180,E1 -4543.216,E2 -4543.216} C_VEL
LIN {X 0,Y 525.921,Z 195.473,A -85,B 0,C 180,E1 -4543.35,E2 -4543.35} C_VEL
LIN {X 0,Y 525.514,Z 274.163,A -85,B 0,C 180,E1 -4544.453,E2 -4544.453} C_VEL
LIN {X 0,Y 525.342,Z 287.054,A -85,B 0,C 180,E1 -4544.784,E2 -4544.784} C_VEL
LIN {X 0,Y 525.142,Z 299.325,A -85,B 0,C 180,E1 -4545.25,E2 -4545.25} C_VEL
LIN {X 0,Y 524.84,Z 311.369,A -85,B 0,C 180,E1 -4545.867,E2 -4545.867} C_VEL
LIN {X 0,Y 524.58,Z 322.53,A -85,B 0,C 180,E1 -4546.612,E2 -4546.612} C_VEL
LIN {X 0,Y 524.338,Z 333.089,A -85,B 0,C 180,E1 -4547.493,E2 -4547.493} C_VEL
LIN {X 0,Y 524.087,Z 341.319,A -85,B 0,C 180,E1 -4548.33,E2 -4548.33} C_VEL
LIN {X 0,Y 523.868,Z 350.079,A -85,B 0,C 180,E1 -4549.409,E2 -4549.409} C_VEL
LIN {X 0,Y 523.671,Z 358.076,A -85,B 0,C 180,E1 -4550.644,E2 -4550.644} C_VEL
LIN {X 0,Y 523.517,Z 364.358,A -85,B 0,C 180,E1 -4551.864,E2 -4551.864} C_VEL
LIN {X 0,Y 523.44,Z 369.954,A -85,B 0,C 180,E1 -4553.282,E2 -4553.282} C_VEL
LIN {X 0,Y 523.323,Z 373.984,A -85,B 0,C 180,E1 -4554.727,E2 -4554.727} C_VEL
LIN {X 0,Y 523.288,Z 375.799,A -85,B 0,C 180,E1 -4555.661,E2 -4555.661} C_VEL
LIN {X 0,Y 523.281,Z 376.973,A -85,B 0,C 180,E1 -4556.588,E2 -4556.588} C_VEL
LIN {X 0,Y 523.272,Z 377.655,A -85,B 0,C 180,E1 -4557.795,E2 -4557.795} C_VEL
LIN {X 0,Y 523.284,Z 377.161,A -85,B 0,C 180,E1 -4559.312,E2 -4559.312} C_VEL
LIN {X 0,Y 523.337,Z 375.13,A -85,B 0,C 180,E1 -4560.798,E2 -4560.798} C_VEL
LIN {X 0,Y 523.359,Z 372.474,A -85,B 0,C 180,E1 -4561.965,E2 -4561.965} C_VEL
LIN {X 0,Y 523.451,Z 368.288,A -85,B 0,C 180,E1 -4563.27,E2 -4563.27} C_VEL
LIN {X 0,Y 523.598,Z 362.759,A -85,B 0,C 180,E1 -4564.563,E2 -4564.563} C_VEL
LIN {X 0,Y 523.686,Z 356.744,A -85,B 0,C 180,E1 -4565.671,E2 -4565.671} C_VEL
LIN {X 0,Y 523.892,Z 348.408,A -85,B 0,C 180,E1 -4566.897,E2 -4566.897} C_VEL
LIN {X 0,Y 524.152,Z 339.543,A -85,B 0,C 180,E1 -4567.949,E2 -4567.949} C_VEL
LIN {X 0,Y 524.375,Z 329.845,A -85,B 0,C 180,E1 -4568.888,E2 -4568.888} C_VEL
LIN {X 0,Y 524.656,Z 318.568,A -85,B 0,C 180,E1 -4569.758,E2 -4569.758} C_VEL
LIN {X 0,Y 524.974,Z 307.288,A -85,B 0,C 180,E1 -4570.447,E2 -4570.447} C_VEL
LIN {X 0,Y 525.155,Z 295.317,A -85,B 0,C 180,E1 -4571.012,E2 -4571.012} C_VEL
LIN {X 0,Y 525.411,Z 282.075,A -85,B 0,C 180,E1 -4571.451,E2 -4571.451} C_VEL
LIN {X 0,Y 525.561,Z 268.551,A -85,B 0,C 180,E1 -4571.731,E2 -4571.731} C_VEL
LIN {X 0,Y 525.926,Z 176.469,A -85,B 0,C 180,E1 -4573.003,E2 -4573.003} C_VEL
LIN {X 0,Y 524.275,Z 167.036,A -85,B 0,C 180,E1 -4573.199,E2 -4573.199} C_VEL
LIN {X 0,Y 524.562,Z 150.738,A -85,B 0,C 180,E1 -4576.242,E2 -4576.242} C_VEL
LIN {X 0,Y 524.681,Z 143.395,A -85,B 0,C 180,E1 -4577.624,E2 -4577.624} C_VEL
LIN {X 0,Y 524.013,Z 138.216,A -85,B 0,C 180,E1 -4578.639,E2 -4578.639} C_VEL
LIN {X 0,Y 523.988,Z 138.212,A -85,B 0,C 180,E1 -4581.516,E2 -4581.516} C_VEL
LIN {X 0,Y 524.068,Z 138.207,A -85,B 0,C 180,E1 -4584.613,E2 -4584.613} C_VEL
LIN {X 0,Y 524.111,Z 138.195,A -85,B 0,C 180,E1 -4587.694,E2 -4587.694} C_VEL
LIN {X 0,Y 524.12,Z 138.197,A -85,B 0,C 180,E1 -4590.768,E2 -4590.768} C_VEL
LIN {X 0,Y 524.005,Z 138.208,A -85,B 0,C 180,E1 -4593.075,E2 -4593.075} C_VEL
LIN {X 0,Y 524.009,Z 138.215,A -85,B 0,C 180,E1 -4596.16,E2 -4596.16} C_VEL
LIN {X 0,Y 523.983,Z 138.21,A -85,B 0,C 180,E1 -4599.262,E2 -4599.262} C_VEL
LIN {X 0,Y 524.002,Z 138.212,A -85,B 0,C 180,E1 -4601.737,E2 -4601.737} C_VEL
LIN {X 0,Y 523.99,Z 138.209,A -85,B 0,C 180,E1 -4605.049,E2 -4605.049} C_VEL
LIN {X 0,Y 523.917,Z 138.227,A -85,B 0,C 180,E1 -4607.971,E2 -4607.971} C_VEL
LIN {X 0,Y 523.953,Z 138.216,A -85,B 0,C 180,E1 -4610.411,E2 -4610.411} C_VEL
LIN {X 0,Y 523.91,Z 138.219,A -85,B 0,C 180,E1 -4612.894,E2 -4612.894} C_VEL
LIN {X 0,Y 523.902,Z 138.224,A -85,B 0,C 180,E1 -4615.422,E2 -4615.422} C_VEL
LIN {X 0,Y 523.909,Z 138.224,A -85,B 0,C 180,E1 -4618.003,E2 -4618.003} C_VEL
LIN {X 0,Y 523.938,Z 138.216,A -85,B 0,C 180,E1 -4620.853,E2 -4620.853} C_VEL
LIN {X 0,Y 523.929,Z 138.224,A -85,B 0,C 180,E1 -4623.729,E2 -4623.729} C_VEL
LIN {X 0,Y 523.9,Z 138.221,A -85,B 0,C 180,E1 -4626.4,E2 -4626.4} C_VEL
LIN {X 0,Y 523.92,Z 138.222,A -85,B 0,C 180,E1 -4629.085,E2 -4629.085} C_VEL
LIN {X 0,Y 523.901,Z 138.221,A -85,B 0,C 180,E1 -4632.124,E2 -4632.124} C_VEL
LIN {X 0,Y 523.937,Z 138.225,A -85,B 0,C 180,E1 -4635.311,E2 -4635.311} C_VEL
LIN {X 0,Y 523.923,Z 138.22,A -85,B 0,C 180,E1 -4638.694,E2 -4638.694} C_VEL
LIN {X 0,Y 523.915,Z 138.219,A -85,B 0,C 180,E1 -4641.898,E2 -4641.898} C_VEL
LIN {X 0,Y 523.921,Z 138.225,A -85,B 0,C 180,E1 -4644.913,E2 -4644.913} C_VEL
LIN {X 0,Y 523.934,Z 138.217,A -85,B 0,C 180,E1 -4647.681,E2 -4647.681} C_VEL
LIN {X 0,Y 523.935,Z 138.222,A -85,B 0,C 180,E1 -4650.681,E2 -4650.681} C_VEL
LIN {X 0,Y 523.906,Z 138.22,A -85,B 0,C 180,E1 -4653.725,E2 -4653.725} C_VEL
LIN {X 0,Y 523.901,Z 138.223,A -85,B 0,C 180,E1 -4656.269,E2 -4656.269} C_VEL
LIN {X 0,Y 523.927,Z 138.226,A -85,B 0,C 180,E1 -4658.766,E2 -4658.766} C_VEL
LIN {X 0,Y 523.93,Z 138.219,A -85,B 0,C 180,E1 -4661.22,E2 -4661.22} C_VEL
LIN {X 0,Y 523.914,Z 138.226,A -85,B 0,C 180,E1 -4664.437,E2 -4664.437} C_VEL
LIN {X 0,Y 523.952,Z 138.214,A -85,B 0,C 180,E1 -4667.607,E2 -4667.607} C_VEL
LIN {X 0,Y 523.932,Z 138.219,A -85,B 0,C 180,E1 -4669.957,E2 -4669.957} C_VEL
LIN {X 0,Y 523.997,Z 138.209,A -85,B 0,C 180,E1 -4673.067,E2 -4673.067} C_VEL
LIN {X 0,Y 523.949,Z 138.215,A -85,B 0,C 180,E1 -4675.384,E2 -4675.384} C_VEL
LIN {X 0,Y 524.107,Z 138.197,A -85,B 0,C 180,E1 -4677.694,E2 -4677.694} C_VEL
LIN {X 0,Y 524.1,Z 138.202,A -85,B 0,C 180,E1 -4680,E2 -4680} C_VEL
LIN {X 0,Y 524.107,Z 138.201,A -85,B 0,C 180,E1 -4682.306,E2 -4682.306} C_VEL
LIN {X 0,Y 524.004,Z 138.215,A -85,B 0,C 180,E1 -4686.16,E2 -4686.16} C_VEL
LIN {X 0,Y 523.948,Z 138.215,A -85,B 0,C 180,E1 -4689.263,E2 -4689.263} C_VEL
LIN {X 0,Y 523.932,Z 138.219,A -85,B 0,C 180,E1 -4692.393,E2 -4692.393} C_VEL
LIN {X 0,Y 523.887,Z 138.228,A -85,B 0,C 180,E1 -4695.563,E2 -4695.563} C_VEL
LIN {X 0,Y 523.907,Z 138.225,A -85,B 0,C 180,E1 -4697.971,E2 -4697.971} C_VEL
LIN {X 0,Y 523.907,Z 138.22,A -85,B 0,C 180,E1 -4700.413,E2 -4700.413} C_VEL
LIN {X 0,Y 523.888,Z 138.223,A -85,B 0,C 180,E1 -4702.895,E2 -4702.895} C_VEL
LIN {X 0,Y 523.883,Z 138.23,A -85,B 0,C 180,E1 -4705.422,E2 -4705.422} C_VEL
LIN {X 0,Y 523.899,Z 138.223,A -85,B 0,C 180,E1 -4708.003,E2 -4708.003} C_VEL
LIN {X 0,Y 523.9,Z 138.222,A -85,B 0,C 180,E1 -4710.846,E2 -4710.846} C_VEL
LIN {X 0,Y 523.914,Z 138.223,A -85,B 0,C 180,E1 -4713.726,E2 -4713.726} C_VEL
LIN {X 0,Y 523.861,Z 138.226,A -85,B 0,C 180,E1 -4716.394,E2 -4716.394} C_VEL
LIN {X 0,Y 523.897,Z 138.228,A -85,B 0,C 180,E1 -4719.087,E2 -4719.087} C_VEL
LIN {X 0,Y 523.893,Z 138.222,A -85,B 0,C 180,E1 -4722.125,E2 -4722.125} C_VEL
LIN {X 0,Y 523.935,Z 138.222,A -85,B 0,C 180,E1 -4725.311,E2 -4725.311} C_VEL
LIN {X 0,Y 523.911,Z 138.224,A -85,B 0,C 180,E1 -4728.696,E2 -4728.696} C_VEL
LIN {X 0,Y 523.897,Z 138.228,A -85,B 0,C 180,E1 -4731.084,E2 -4731.084} C_VEL
LIN {X 0,Y 523.855,Z 138.226,A -85,B 0,C 180,E1 -4733.821,E2 -4733.821} C_VEL
LIN {X 0,Y 523.897,Z 138.227,A -85,B 0,C 180,E1 -4736.632,E2 -4736.632} C_VEL
LIN {X 0,Y 523.908,Z 138.223,A -85,B 0,C 180,E1 -4739.352,E2 -4739.352} C_VEL
LIN {X 0,Y 523.912,Z 138.225,A -85,B 0,C 180,E1 -4742.295,E2 -4742.295} C_VEL
LIN {X 0,Y 523.892,Z 138.228,A -85,B 0,C 180,E1 -4745.426,E2 -4745.426} C_VEL
LIN {X 0,Y 523.922,Z 138.363,A -85,B 0,C 180,E1 -4745.897,E2 -4745.897} C_VEL
LIN {X 0,Y 525.235,Z 145.727,A -85,B 0,C 180,E1 -4747.167,E2 -4747.167} C_VEL
LIN {X 0,Y 524.967,Z 160.964,A -85,B 0,C 180,E1 -4749.63,E2 -4749.63} C_VEL
LIN {X 0,Y 524.568,Z 177.465,A -85,B 0,C 180,E1 -4752.254,E2 -4752.254} C_VEL
LIN {X 0,Y 524.248,Z 193.943,A -85,B 0,C 180,E1 -4754.846,E2 -4754.846} C_VEL
LIN {X 0,Y 525.911,Z 205.083,A -85,B 0,C 180,E1 -4755.05,E2 -4755.05} C_VEL
LIN {X 0,Y 525.464,Z 302.594,A -85,B 0,C 180,E1 -4756.414,E2 -4756.414} C_VEL
LIN {X 0,Y 525.25,Z 316.438,A -85,B 0,C 180,E1 -4756.778,E2 -4756.778} C_VEL
LIN {X 0,Y 524.995,Z 329.362,A -85,B 0,C 180,E1 -4757.288,E2 -4757.288} C_VEL
LIN {X 0,Y 524.665,Z 341.975,A -85,B 0,C 180,E1 -4757.971,E2 -4757.971} C_VEL
LIN {X 0,Y 524.412,Z 353.763,A -85,B 0,C 180,E1 -4758.795,E2 -4758.795} C_VEL
LIN {X 0,Y 524.122,Z 364.686,A -85,B 0,C 180,E1 -4759.766,E2 -4759.766} C_VEL
LIN {X 0,Y 523.88,Z 373.559,A -85,B 0,C 180,E1 -4760.736,E2 -4760.736} C_VEL
LIN {X 0,Y 523.691,Z 382.214,A -85,B 0,C 180,E1 -4761.899,E2 -4761.899} C_VEL
LIN {X 0,Y 523.51,Z 389.123,A -85,B 0,C 180,E1 -4763.06,E2 -4763.06} C_VEL
LIN {X 0,Y 523.49,Z 394.663,A -85,B 0,C 180,E1 -4764.221,E2 -4764.221} C_VEL
LIN {X 0,Y 523.355,Z 399.003,A -85,B 0,C 180,E1 -4765.379,E2 -4765.379} C_VEL
LIN {X 0,Y 523.443,Z 401.304,A -85,B 0,C 180,E1 -4766.151,E2 -4766.151} C_VEL
LIN {X 0,Y 523.367,Z 403.165,A -85,B 0,C 180,E1 -4766.921,E2 -4766.921} C_VEL
LIN {X 0,Y 523.335,Z 404.561,A -85,B 0,C 180,E1 -4767.691,E2 -4767.691} C_VEL
LIN {X 0,Y 523.253,Z 406.162,A -85,B 0,C 180,E1 -4769.23,E2 -4769.23} C_VEL
LIN {X 0,Y 523.251,Z 406.377,A -85,B 0,C 180,E1 -4770,E2 -4770} C_VEL
LIN {X 0,Y 523.275,Z 405.551,A -85,B 0,C 180,E1 -4771.539,E2 -4771.539} C_VEL
LIN {X 0,Y 523.335,Z 404.555,A -85,B 0,C 180,E1 -4772.309,E2 -4772.309} C_VEL
LIN {X 0,Y 523.367,Z 403.156,A -85,B 0,C 180,E1 -4773.079,E2 -4773.079} C_VEL
LIN {X 0,Y 523.422,Z 400.216,A -85,B 0,C 180,E1 -4774.235,E2 -4774.235} C_VEL
LIN {X 0,Y 523.456,Z 396.234,A -85,B 0,C 180,E1 -4775.393,E2 -4775.393} C_VEL
LIN {X 0,Y 523.502,Z 391.067,A -85,B 0,C 180,E1 -4776.561,E2 -4776.561} C_VEL
LIN {X 0,Y 523.628,Z 384.653,A -85,B 0,C 180,E1 -4777.713,E2 -4777.713} C_VEL
LIN {X 0,Y 523.794,Z 376.603,A -85,B 0,C 180,E1 -4778.876,E2 -4778.876} C_VEL
LIN {X 0,Y 524.006,Z 368.396,A -85,B 0,C 180,E1 -4779.846,E2 -4779.846} C_VEL
LIN {X 0,Y 524.318,Z 358.387,A -85,B 0,C 180,E1 -4780.816,E2 -4780.816} C_VEL
LIN {X 0,Y 524.588,Z 347.162,A -85,B 0,C 180,E1 -4781.685,E2 -4781.685} C_VEL
LIN {X 0,Y 524.845,Z 335.98,A -85,B 0,C 180,E1 -4782.372,E2 -4782.372} C_VEL
LIN {X 0,Y 525.129,Z 323.677,A -85,B 0,C 180,E1 -4782.954,E2 -4782.954} C_VEL
LIN {X 0,Y 525.362,Z 310.666,A -85,B 0,C 180,E1 -4783.391,E2 -4783.391} C_VEL
LIN {X 0,Y 525.543,Z 296.78,A -85,B 0,C 180,E1 -4783.682,E2 -4783.682} C_VEL
LIN {X 0,Y 525.783,Z 203.79,A -85,B 0,C 180,E1 -4784.97,E2 -4784.97} C_VEL
LIN {X 0,Y 524.226,Z 193.647,A -85,B 0,C 180,E1 -4785.174,E2 -4785.174} C_VEL
LIN {X 0,Y 524.616,Z 174.755,A -85,B 0,C 180,E1 -4788.128,E2 -4788.128} C_VEL
LIN {X 0,Y 525.084,Z 154.149,A -85,B 0,C 180,E1 -4791.391,E2 -4791.391} C_VEL
LIN {X 0,Y 525.175,Z 145.163,A -85,B 0,C 180,E1 -4792.836,E2 -4792.836} C_VEL
LIN {X 0,Y 523.903,Z 138.227,A -85,B 0,C 180,E1 -4794.056,E2 -4794.056} C_VEL
LIN {X 0,Y 523.892,Z 138.23,A -85,B 0,C 180,E1 -4797.137,E2 -4797.137} C_VEL
LIN {X 0,Y 523.867,Z 138.231,A -85,B 0,C 180,E1 -4799.761,E2 -4799.761} C_VEL
LIN {X 0,Y 523.896,Z 138.225,A -85,B 0,C 180,E1 -4802.452,E2 -4802.452} C_VEL
LIN {X 0,Y 523.88,Z 138.232,A -85,B 0,C 180,E1 -4805.23,E2 -4805.23} C_VEL
LIN {X 0,Y 523.876,Z 138.225,A -85,B 0,C 180,E1 -4808.106,E2 -4808.106} C_VEL
LIN {X 0,Y 523.878,Z 138.23,A -85,B 0,C 180,E1 -4811.3,E2 -4811.3} C_VEL
LIN {X 0,Y 523.933,Z 138.222,A -85,B 0,C 180,E1 -4814.688,E2 -4814.688} C_VEL
LIN {X 0,Y 523.888,Z 138.223,A -85,B 0,C 180,E1 -4817.875,E2 -4817.875} C_VEL
LIN {X 0,Y 523.892,Z 138.229,A -85,B 0,C 180,E1 -4821.085,E2 -4821.085} C_VEL
LIN {X 0,Y 523.855,Z 138.225,A -85,B 0,C 180,E1 -4823.822,E2 -4823.822} C_VEL
LIN {X 0,Y 523.897,Z 138.228,A -85,B 0,C 180,E1 -4826.632,E2 -4826.632} C_VEL
LIN {X 0,Y 523.909,Z 138.221,A -85,B 0,C 180,E1 -4829.353,E2 -4829.353} C_VEL
LIN {X 0,Y 523.914,Z 138.221,A -85,B 0,C 180,E1 -4832.296,E2 -4832.296} C_VEL
LIN {X 0,Y 523.894,Z 138.22,A -85,B 0,C 180,E1 -4835.426,E2 -4835.426} C_VEL
